// ---- VISUs/Behelyezes.TcVIS
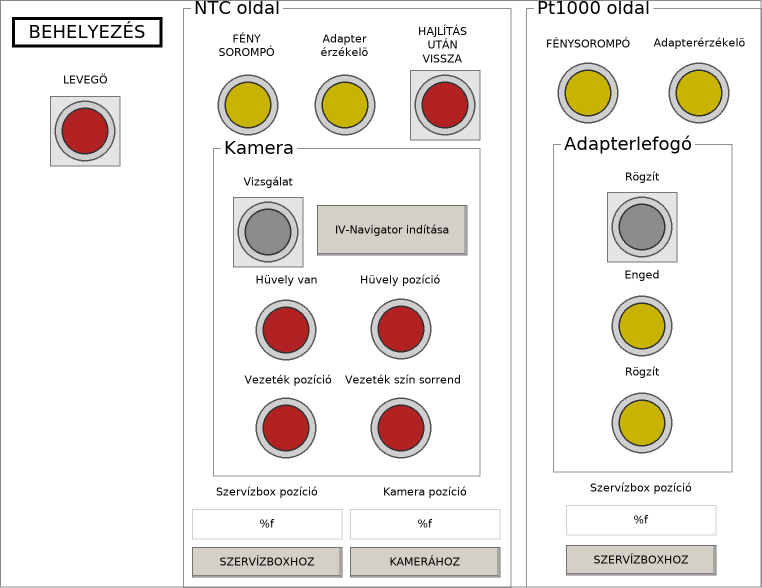
VISUALIZATION Behelyezes  // 762x588
    GroupBox (526,0 236x587), "Pt1000 oldal"
        GroupBox (27,136 179x336), "Adapterlefogó"
            PushSwitch (54,56 70x70), variable: GVL.bAdapterLefogo, behaviour: TOGGLE, style: Switch-PushSwitch-Gray
            Lamp1 (54,155 70x70), variable: GVL.bAdapterLefogoBent, style: Lamp-Lamp1-Yellow
            Lamp1 (54,252 70x70), variable: GVL.bAdapterLefogoKint, style: Lamp-Lamp1-Yellow
            Label (61,226 57x20), "Rögzít"
            Label (62,129 54x20), "Enged"
            Label (60,31 59x20), "Rögzít"
        Lamp1 (138,58 70x70), variable: GVL.bAdaptererzekelo, style: Lamp-Lamp1-Yellow
        Label (122,33 103x20), "Adapterérzékelö"
        Lamp1 (27,58 70x70), variable: GVL.bFenysorompoPt, style: Lamp-Lamp1-Yellow
        Label (10,34 104x20), "FÉNYSOROMPÓ"
        Group (40,478 150x97)
            Button (0,67 150x30), "SZERVÍZBOXHOZ"
                OnMouseUp: execute { PISTITENGELY.lrPistiPosition:=GVL.lrPtSzervizbox; PISTITENGELY.sPistiAxisCommand:='MOVE'; }
            Textfield (0,27 150x30), "%f", text variable: GVL.lrPtSzervizbox
                OnMouseClick: write the text variable via VisuDialogs.Numpad, min -10000, max -1
            Label (0,0 150x20), "Szervízbox pozíció"
    RoundedRectangle (12,17 150x30)
    Label (12,17 150x30), "BEHELYEZÉS"
    GroupBox (183,0 328x588), "NTC oldal"
        GroupBox (30,140 267x336), "Kamera"
            Group (20,32 70x95)
                PushSwitch (0,25 70x70), variable: GVL.bKameraTrigger, behaviour: TOGGLE, style: Switch-PushSwitch-Gray
                Label (2,0 67x20), "Vizsgálat"
            Lamp1 (153,154 70x70), variable: GVL.bKameraHulsePozOK, style: Lamp-Lamp1-Green
            Lamp1 (153,253 70x70), variable: GVL.bKameraSzinekOK, style: Lamp-Lamp1-Green
            Label (130,230 120x20), "Vezeték szín sorrend"
            Label (140,130 94x20), "Hüvely pozíció"
            Lamp1 (153,154 70x70), variable: NOT GVL.bKameraHulsePozOK, invisible if: NOT KAMERA.bVizsgalatKesz OR GVL.bKameraHulsePozOK, style: Lamp-Lamp1-Red
            Lamp1 (153,253 70x70), variable: NOT GVL.bKameraSzinekOK, invisible if: NOT KAMERA.bVizsgalatKesz OR GVL.bKameraSzinekOK, style: Lamp-Lamp1-Red
            Label (30,230 90x20), "Vezeték pozíció"
            Lamp1 (38,253 70x70), variable: GVL.bKameraVezetekPozOK, style: Lamp-Lamp1-Green
            Lamp1 (38,253 70x70), variable: NOT GVL.bKameraVezetekPozOK, invisible if: NOT KAMERA.bVizsgalatKesz OR GVL.bKameraVezetekPozOK, style: Lamp-Lamp1-Red
            Button (104,65 150x50), "IV-Navigator indítása", tooltip "A jelölö lézer saját vezérlö szoftvere", pressed state: Laser.bStartFOBADraw
                OnMouseUp: execute { KAMERA.bStartIVNav:=TRUE; }
            Label (32,130 83x20), "Hüvely van"
            Lamp1 (38,155 70x70), variable: GVL.bKameraHulseVanOK, style: Lamp-Lamp1-Green
            Lamp1 (38,155 70x70), variable: NOT GVL.bKameraHulseVanOK, invisible if: NOT KAMERA.bVizsgalatKesz OR GVL.bKameraHulseVanOK, style: Lamp-Lamp1-Red
        Group (9,482 150x95)
            Textfield (0,27 150x30), "%f", text variable: GVL.lrNTCSzervizbox
                OnMouseClick: write the text variable via VisuDialogs.Numpad, min -10000, max -1
            Button (0,65 150x30), "SZERVÍZBOXHOZ"
                OnMouseUp: execute { JOZSITENGELY.lrJozsiPosition:=GVL.lrNTCSzervizbox; JOZSITENGELY.sJozsiAxisCommand:='MOVE'; }
            Label (0,0 150x20), "Szervízbox pozíció"
        Lamp1 (30,70 70x70), variable: GVL.bFenysorompoNTC, style: Lamp-Lamp1-Yellow
        Label (10,30 107x31), "FÉNY SOROMPÓ"
        Group (167,482 150x95)
            Textfield (0,27 150x30), "%f", text variable: GVL.lrNTCKameraPosition
                OnMouseClick: write the text variable via VisuDialogs.Numpad, min -10000, max -1
            Button (0,65 150x30), "KAMERÁHOZ"
                OnMouseUp: execute { JOZSITENGELY.lrJozsiPosition:=GVL.lrNTCKameraPosition; JOZSITENGELY.sJozsiAxisCommand:='MOVE'; }
            Label (0,0 150x20), "Kamera pozíció"
        Label (110,30 103x31), "Adapter érzékelö"
        Label (220,20 79x50), "HAJLÍTÁS UTÁN VISSZA"
    Label (51,70 69x20), "LEVEGÖ"
    PushSwitch (50,96 70x70), variable: MAIN.bLevego, behaviour: TOGGLE, style: Switch-PushSwitch-Red
    Lamp1 (310,70 70x70), variable: GVL.bNTCAdapterErzekelo, style: Lamp-Lamp1-Yellow
    PushSwitch (410,70 70x70), variable: AUTOMATA.bHajlitasUtanVissza, behaviour: TOGGLE, style: Switch-PushSwitch-Red
END_VISUALIZATION

// ---- VISUs/Rendszerinditas.TcVIS
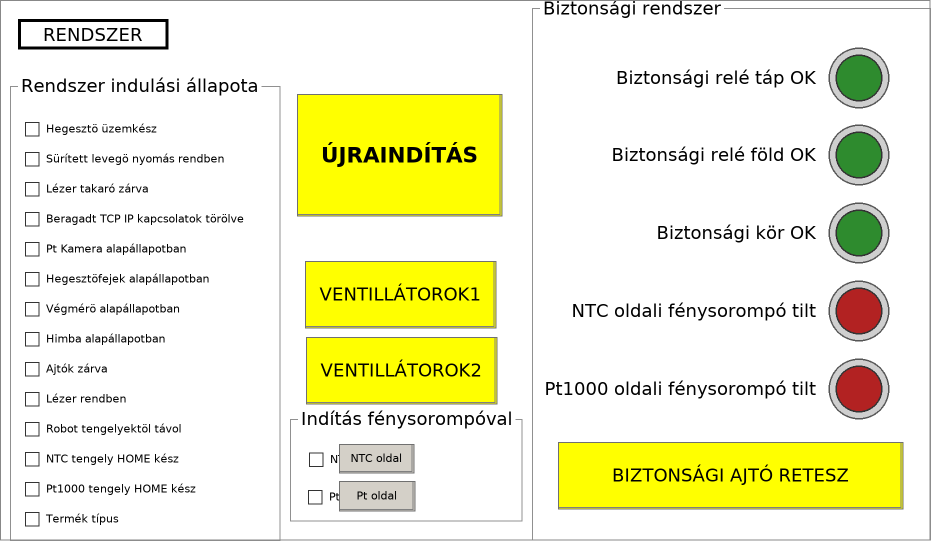
VISUALIZATION Rendszerinditas  // 931x541
    RoundedRectangle (18,19 150x30)
    Label (18,20 150x30), "RENDSZER"
    Button (297,94 205x122), "ÚJRAINDÍTÁS"
        OnMouseUp: execute { INIT.bRestart:=TRUE; }
    GroupBox (10,78 270x463), "Rendszer indulási állapota"
        Frame (13,36 239x351)
            shows Start_ellenorzes()
    GroupBox (532,0 399x540), "Biztonsági rendszer"
        Button (26,442 345x67), "BIZTONSÁGI AJTÓ RETESZ", pressed state: GVL.bBiztonsagiZarBe
            OnMouseClick: execute {
                IF GVL.bBiztonsagiZarBe=TRUE THEN
                	WHILE NOT (ROBOTREMOTE.sRobotCommand='') DO
                		;
                	END_WHILE
                	ROBOTREMOTE.sRobotCommand := 'Pause';
                	ROBOTREMOTE.bRobotCommandSend := TRUE;
                ELSE
                	WHILE NOT (ROBOTREMOTE.sRobotCommand='') DO
                		;
                	END_WHILE
                	ROBOTREMOTE.sRobotCommand := 'Continue';
                	ROBOTREMOTE.bRobotCommandSend := TRUE;
                END_IF
                GVL.bBiztonsagiZarBe:=NOT GVL.bBiztonsagiZarBe;
            }
        Lamp1 (292,43 70x70), variable: GVL.bBiztonsagiTap, style: Lamp-Lamp1-Green
        Label (17,63 270x30), "Biztonsági relé táp OK"
        Lamp1 (292,120 70x70), variable: NOT GVL.bBiztonsagiFold, style: Lamp-Lamp1-Green
        Label (17,140 270x30), "Biztonsági relé föld OK"
        Lamp1 (292,198 70x70), variable: (GVL.bBiztonsagiTap AND NOT GVL.bBiztonsagiFold) OR (NOT GVL.bBiztonsagiTap AND GVL.bBiztonsagiFold), style: Lamp-Lamp1-Green
        Label (17,218 270x30), "Biztonsági kör OK"
        Lamp1 (292,276 70x70), variable: NOT GVL.bFenysorompoNTC, style: Lamp-Lamp1-Red
        Label (17,296 270x30), "NTC oldali fénysorompó tilt"
        Lamp1 (292,354 70x70), variable: NOT GVL.bFenysorompoPt, style: Lamp-Lamp1-Red
        Label (17,374 270x30), "Pt1000 oldali fénysorompó tilt"
    Button (305,261 191x67), "VENTILLÁTOROK1", pressed state: GVL.bVentillatorok1Be
        toggle GVL.bVentillatorok1Be
    Button (306,337 191x67), "VENTILLÁTOROK2", pressed state: GVL.bVentillatorok2Be
        toggle GVL.bVentillatorok2Be
    GroupBox (290,411 232x110), "Indítás fénysorompóval"
        Checkbox (16,71 95x30), "Pt oldal", variable: GVL.bPtInditasFenysorompoval, input disabled if: TRUE
        Checkbox (17,34 94x29), "NTC oldal", variable: GVL.bNTCInditasFenysorompoval, input disabled if: TRUE
        Button (49,33 75x29), "NTC oldal", pressed state: GVL.bNTCInditasFenysorompoval
            toggle GVL.bNTCInditasFenysorompoval
            OnMouseUp: execute { AUTOMATA.iState:=102; }
        Button (49,70 76x30), "Pt oldal", pressed state: GVL.bPtInditasFenysorompoval
            toggle GVL.bPtInditasFenysorompoval
            OnMouseUp: execute { AUTOMATA.iState2:=103; }
END_VISUALIZATION

// ---- VISUs/Start_ellenorzes.TcVIS
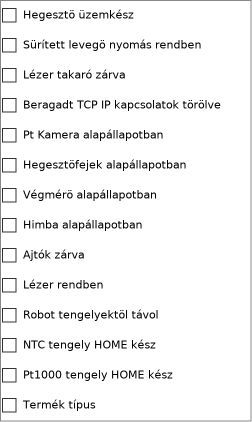
VISUALIZATION Start_ellenorzes  // 252x422
    Checkbox (0,30 250x30), "Sürített levegö nyomás rendben", variable: MAIN.bLevegoOK
    Checkbox (0,90 250x30), "Beragadt TCP IP kapcsolatok törölve", variable: INIT.bTCPKesz
    Checkbox (0,150 250x30), "Hegesztöfejek alapállapotban", variable: INIT.bHegesztoFejekKesz
    Checkbox (0,180 250x30), "Végmérö alapállapotban", variable: INIT.bVegmeroKesz
    Checkbox (0,300 250x30), "Robot tengelyektöl távol", variable: INIT.bRobotKesz
    Checkbox (0,270 250x30), "Lézer rendben", variable: INIT.bLezerKesz
    Checkbox (0,330 250x30), "NTC tengely HOME kész", variable: INIT.bNTCTengelyKesz
    Checkbox (0,360 250x30), "Pt1000 tengely HOME kész", variable: INIT.bPt1000TengelyKesz
    Checkbox (0,60 250x30), "Lézer takaró zárva", variable: VEGMERO.bLezertakaroZarva
    Checkbox (0,0 250x30), "Hegesztö üzemkész", variable: INIT.bHegesztoKesz
    Checkbox (0,390 250x30), "Termék típus", variable: GVL.bProductTypeOK
    Checkbox (0,240 250x30), "Ajtók zárva", variable: NOT GVL.bBiztonsagiFold AND GVL.bBiztonsagiTap
    Checkbox (0,210 250x30), "Himba alapállapotban", variable: INIT.bHimbaKesz
    Checkbox (0,120 250x30), "Pt Kamera alapállapotban", variable: INIT.bKameraKesz
END_VISUALIZATION

// ---- VISUs/Tengely_NTC_beallitasok.TcVIS
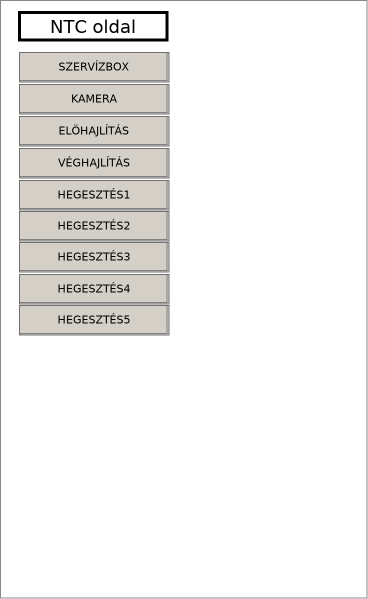
VISUALIZATION Tengely_NTC_beallitasok  // 368x599
    Label (297,567 69x30)
    RoundedRectangle (18,11 150x30)
    Label (18,12 150x30), "NTC oldal"
    Button (19,116 150x30), "ELÖHAJLÍTÁS"
        OnMouseUp: execute { GVL.iFoLapozo:=GVL.SZERVIZ_FUL; GVL.iSzervizLapozo:=GVL.HAJLITOK_FUL; }
    Button (19,148 150x30), "VÉGHAJLÍTÁS"
        OnMouseUp: execute { GVL.iFoLapozo:=GVL.SZERVIZ_FUL; GVL.iSzervizLapozo:=GVL.HAJLITOK_FUL; }
    Button (19,180 150x30), "HEGESZTÉS1"
        OnMouseUp: execute {
            GVL.iFoLapozo:=GVL.SZERVIZ_FUL;
            GVL.iSzervizLapozo:=GVL.HEGESZTES_FUL;
            GVL.iTengelyLapozo:=GVL.NTC_TENGELY_FUL;
        }
    Button (19,211 150x30), "HEGESZTÉS2"
        OnMouseUp: execute {
            GVL.iFoLapozo:=GVL.SZERVIZ_FUL;
            GVL.iSzervizLapozo:=GVL.HEGESZTES_FUL;
            GVL.iTengelyLapozo:=GVL.NTC_TENGELY_FUL;
        }
    Button (19,242 150x30), "HEGESZTÉS3"
        OnMouseUp: execute {
            GVL.iFoLapozo:=GVL.SZERVIZ_FUL;
            GVL.iSzervizLapozo:=GVL.HEGESZTES_FUL;
            GVL.iTengelyLapozo:=GVL.NTC_TENGELY_FUL;
        }
    Button (19,274 150x30), "HEGESZTÉS4"
        OnMouseUp: execute {
            GVL.iFoLapozo:=GVL.SZERVIZ_FUL;
            GVL.iSzervizLapozo:=GVL.HEGESZTES_FUL;
            GVL.iTengelyLapozo:=GVL.NTC_TENGELY_FUL;
        }
    Button (19,305 150x30), "HEGESZTÉS5"
        OnMouseUp: execute {
            GVL.iFoLapozo:=GVL.SZERVIZ_FUL;
            GVL.iSzervizLapozo:=GVL.HEGESZTES_FUL;
            GVL.iTengelyLapozo:=GVL.NTC_TENGELY_FUL;
        }
    Button (19,52 150x30), "SZERVÍZBOX"
        OnMouseUp: execute { GVL.iFoLapozo:=GVL.SZERVIZ_FUL; GVL.iSzervizLapozo:=GVL.BEHELYEZES_FUL; }
    Button (19,84 150x30), "KAMERA"
        OnMouseUp: execute { GVL.iFoLapozo:=GVL.SZERVIZ_FUL; GVL.iSzervizLapozo:=GVL.BEHELYEZES_FUL; }
END_VISUALIZATION

// ---- VISUs/Tengely_Pt1000.TcVIS
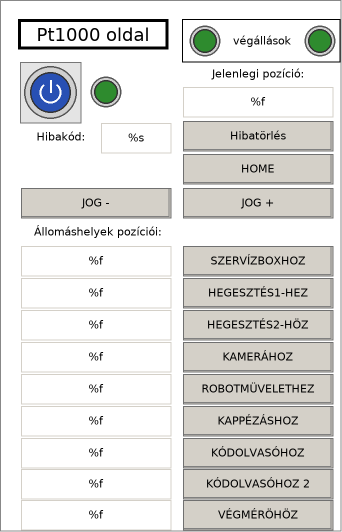
VISUALIZATION Tengely_Pt1000  // 342x532
    PowerSwitch (20,62 61x61), variable: GVL.bPistiServo, behaviour: TOGGLE, style: Switch-PowerSwitch-Blue
    Button (183,154 150x30), "HOME"
        OnMouseUp: execute { PISTITENGELY.sPistiAxisCommand:='HOME'; }
    Button (183,188 150x30), "JOG +"
        tap PISTITENGELY.bPistiJOGPlus
    Button (21,188 150x30), "JOG -"
        tap PISTITENGELY.bPistiJOGMinus
    Button (183,121 150x30), "Hibatörlés"
        tap PISTITENGELY.bPistiReset
    Textfield (101,123 70x30), "%s", text variable: PISTITENGELY.nPistiErrorCode, input disabled if: TRUE
    Textfield (21,310 150x30), "%f", text variable: GVL.lrHegesztoPosition7
    Button (183,310 150x30), "HEGESZTÉS2-HÖZ"
        OnMouseUp: execute { PISTITENGELY.lrPistiPosition:=GVL.lrHegesztoPosition7; PISTITENGELY.sPistiAxisCommand:='MOVE'; }
    Label (183,64 150x20), "Jelenlegi pozíció:"
    Textfield (183,87 150x30), "%f", text variable: PISTITENGELY.lrPistiActPos, input disabled if: TRUE
    Button (183,246 150x30), "SZERVÍZBOXHOZ"
        OnMouseUp: execute { PISTITENGELY.lrPistiPosition:=GVL.lrPtSzervizbox; PISTITENGELY.sPistiAxisCommand:='MOVE'; }
    Textfield (21,246 150x30), "%f", text variable: GVL.lrPtSzervizbox
    Textfield (21,278 150x30), "%f", text variable: GVL.lrHegesztoPosition6
    Button (183,278 150x30), "HEGESZTÉS1-HEZ"
        OnMouseUp: execute { PISTITENGELY.lrPistiPosition:=GVL.lrHegesztoPosition6; PISTITENGELY.sPistiAxisCommand:='MOVE'; }
    Lamp1 (88,74 36x36), variable: PISTITENGELY.bHomeReady, style: Lamp-Lamp1-Green
    RoundedRectangle (18,19 150x30)
    Label (18,20 150x30), "Pt1000 oldal"
    Textfield (21,374 150x30), "%f", text variable: GVL.lrRobotKappePosition
    Button (183,374 150x30), "ROBOTMÜVELETHEZ"
        OnMouseUp: execute { PISTITENGELY.lrPistiPosition:=GVL.lrRobotKappePosition; PISTITENGELY.sPistiAxisCommand:='MOVE'; }
    Textfield (21,500 150x30), "%f", text variable: GVL.lrVegmeroPosition
    Button (183,500 150x30), "VÉGMÉRÖHÖZ"
        OnMouseUp: execute { PISTITENGELY.lrPistiPosition:=GVL.lrVegmeroPosition; PISTITENGELY.sPistiAxisCommand:='MOVE'; }
    Textfield (21,406 150x30), "%f", text variable: GVL.lrKappePosition
    Button (183,406 150x30), "KAPPÉZÁSHOZ"
        OnMouseUp: execute { PISTITENGELY.lrPistiPosition:=GVL.lrKappePosition; PISTITENGELY.sPistiAxisCommand:='MOVE'; }
    Textfield (21,438 150x30), "%f", text variable: GVL.lrKodolvasasPosition
    Button (183,438 150x30), "KÓDOLVASÓHOZ"
        OnMouseUp: execute { PISTITENGELY.lrPistiPosition:=GVL.lrKodolvasasPosition; PISTITENGELY.sPistiAxisCommand:='MOVE'; }
    Label (26,127 70x20), "Hibakód:"
    Label (23,222 150x20), "Állomáshelyek pozíciói:"
    Group (182,19 158x43)
        Rectangle (0,0 158x43)
        Lamp1 (5,4 36x36), variable: GVL.bPistiNegSwitch, style: Lamp-Lamp1-Green
        Lamp1 (120,4 36x36), variable: GVL.bPistiPosSwitch, style: Lamp-Lamp1-Green
        Label (45,12 70x20), "végállások"
    Textfield (21,342 150x30), "%f", text variable: GVL.lrPtKameraPosition
    Button (183,342 150x30), "KAMERÁHOZ"
        OnMouseUp: execute { PISTITENGELY.lrPistiPosition:=GVL.lrPtKameraPosition; PISTITENGELY.sPistiAxisCommand:='MOVE'; }
    Textfield (21,469 150x30), "%f", text variable: GVL.lrKodolvasasPosition2
    Button (183,469 150x30), "KÓDOLVASÓHOZ 2"
        OnMouseUp: execute { PISTITENGELY.lrPistiPosition:=GVL.lrKodolvasasPosition2; PISTITENGELY.sPistiAxisCommand:='MOVE'; }
END_VISUALIZATION

// ---- VISUs/Tengelyek.TcVIS
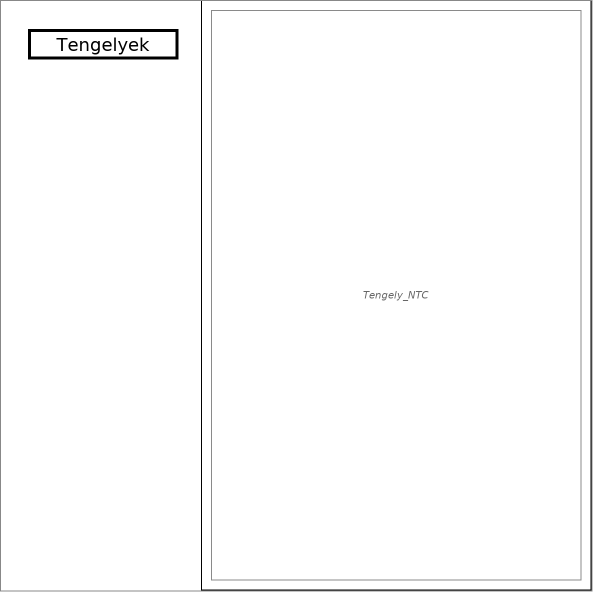
VISUALIZATION Tengelyek  // 593x592
    Group (201,0 390x590)
        Rectangle (0,0 390x590)
        TabControl (10,10 370x570)
            shows Tengely_NTC()
            shows Tengely_Pt1000()
            [0]: TabTitle=NTC oldal
            [1]: TabTitle=Pt1000 oldal
    RoundedRectangle (28,29 150x30)
    Label (28,30 150x30), "Tengelyek"
END_VISUALIZATION

// ---- VISUs/Tengely_NTC.TcVIS
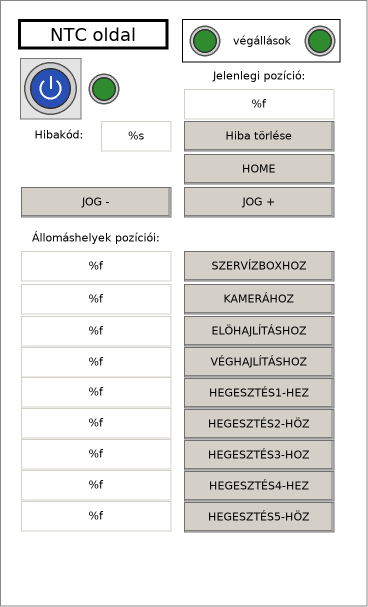
VISUALIZATION Tengely_NTC  // 368x607
    PowerSwitch (20,58 61x61), variable: GVL.bJozsiServo, behaviour: TOGGLE, style: Switch-PowerSwitch-Blue
    Button (184,154 150x30), "HOME"
        OnMouseUp: execute { JOZSITENGELY.sJozsiAxisCommand:='HOME'; }
    Button (184,187 150x30), "JOG +"
        tap JOZSITENGELY.bJozsiJOGPlus
    Button (21,187 150x30), "JOG -"
        tap JOZSITENGELY.bJozsiJOGMinus
    Button (184,121 150x30), "Hiba törlése"
        tap JOZSITENGELY.bJozsiReset
    Textfield (101,121 70x30), "%s", text variable: JOZSITENGELY.nJozsiErrorCode, input disabled if: TRUE
    Textfield (21,316 150x30), "%f", text variable: GVL.lrHajlitoPosition1
    Button (184,316 150x30), "ELÖHAJLÍTÁSHOZ"
        OnMouseUp: execute { JOZSITENGELY.lrJozsiPosition:=GVL.lrHajlitoPosition1; JOZSITENGELY.sJozsiAxisCommand:='MOVE'; }
    Textfield (184,89 150x30), "%f", text variable: JOZSITENGELY.lrJozsiActPos, input disabled if: TRUE
    Label (184,66 150x20), "Jelenlegi pozíció:"
    Textfield (21,284 150x30), "%f", text variable: GVL.lrNTCKameraPosition
    Button (184,284 150x30), "KAMERÁHOZ"
        OnMouseUp: execute { JOZSITENGELY.lrJozsiPosition:=GVL.lrNTCKameraPosition; JOZSITENGELY.sJozsiAxisCommand:='MOVE'; }
    Textfield (21,377 150x30), "%f", text variable: GVL.lrHegesztoPosition1
    Button (184,378 150x30), "HEGESZTÉS1-HEZ"
        OnMouseUp: execute { JOZSITENGELY.lrJozsiPosition:=GVL.lrHegesztoPosition1; JOZSITENGELY.sJozsiAxisCommand:='MOVE'; }
    Textfield (21,408 150x30), "%f", text variable: GVL.lrHegesztoPosition2
    Button (184,409 150x30), "HEGESZTÉS2-HÖZ"
        OnMouseUp: execute { JOZSITENGELY.lrJozsiPosition:=GVL.lrHegesztoPosition2; JOZSITENGELY.sJozsiAxisCommand:='MOVE'; }
    Textfield (21,439 150x30), "%f", text variable: GVL.lrHegesztoPosition3
    Button (184,440 150x30), "HEGESZTÉS3-HOZ"
        OnMouseUp: execute { JOZSITENGELY.lrJozsiPosition:=GVL.lrHegesztoPosition3; JOZSITENGELY.sJozsiAxisCommand:='MOVE'; }
    Textfield (21,470 150x30), "%f", text variable: GVL.lrHegesztoPosition4
    Button (184,471 150x30), "HEGESZTÉS4-HEZ"
        OnMouseUp: execute { JOZSITENGELY.lrJozsiPosition:=GVL.lrHegesztoPosition4; JOZSITENGELY.sJozsiAxisCommand:='MOVE'; }
    Textfield (21,501 150x30), "%f", text variable: GVL.lrHegesztoPosition5
    Button (184,502 150x30), "HEGESZTÉS5-HÖZ"
        OnMouseUp: execute { JOZSITENGELY.lrJozsiPosition:=GVL.lrHegesztoPosition5; JOZSITENGELY.sJozsiAxisCommand:='MOVE'; }
    Label (297,575 69x30)
    Button (184,251 150x30), "SZERVÍZBOXHOZ"
        OnMouseUp: execute { JOZSITENGELY.lrJozsiPosition:=GVL.lrNTCSzervizbox; JOZSITENGELY.sJozsiAxisCommand:='MOVE'; }
    Lamp1 (86,71 36x36), variable: JOZSITENGELY.bHomeReady, style: Lamp-Lamp1-Green
    Label (24,125 70x20), "Hibakód:"
    Label (21,228 150x20), "Állomáshelyek pozíciói:"
    RoundedRectangle (18,19 150x30)
    Label (18,20 150x30), "NTC oldal"
    Group (182,19 158x43)
        Rectangle (0,0 158x43)
        Lamp1 (5,4 36x36), variable: GVL.bJozsiNegSwitch, style: Lamp-Lamp1-Green
        Lamp1 (120,4 36x36), variable: GVL.bJozsiPosSwitch, style: Lamp-Lamp1-Green
        Label (45,12 70x20), "végállások"
    Textfield (21,251 150x30), "%f", text variable: GVL.lrNTCSzervizbox
    Textfield (21,347 150x30), "%f", text variable: GVL.lrHajlitoPosition2
    Button (184,347 150x30), "VÉGHAJLÍTÁSHOZ"
        OnMouseUp: execute { JOZSITENGELY.lrJozsiPosition:=GVL.lrHajlitoPosition2; JOZSITENGELY.sJozsiAxisCommand:='MOVE'; }
END_VISUALIZATION

// ---- VISUs/Tengely_Pt1000_beallitasok.TcVIS
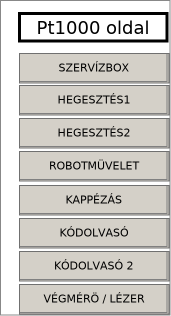
VISUALIZATION Tengely_Pt1000_beallitasok  // 171x316
    RoundedRectangle (18,12 150x30)
    Label (18,13 150x30), "Pt1000 oldal"
    Button (19,118 150x30), "HEGESZTÉS2"
        OnMouseUp: execute { GVL.iFoLapozo:=GVL.SZERVIZ_FUL; GVL.iSzervizLapozo:=GVL.HEGESZTES_FUL; }
    Button (19,53 150x30), "SZERVÍZBOX"
        OnMouseUp: execute {
            GVL.iFoLapozo:=GVL.SZERVIZ_FUL;
            GVL.iSzervizLapozo:=GVL.BEHELYEZES_FUL;
            GVL.iTengelyLapozo:=GVL.PT_TENGELY_FUL;
        }
    Button (19,85 150x30), "HEGESZTÉS1"
        OnMouseUp: execute { GVL.iFoLapozo:=GVL.SZERVIZ_FUL; GVL.iSzervizLapozo:=GVL.HEGESZTES_FUL; }
    Button (19,151 150x30), "ROBOTMÜVELET"
        OnMouseUp: execute { GVL.iFoLapozo:=GVL.SZERVIZ_FUL; GVL.iSzervizLapozo:=GVL.ROBOT_FUL; }
    Button (19,284 150x30), "VÉGMÉRÖ / LÉZER"
        OnMouseUp: execute { GVL.iFoLapozo:=GVL.SZERVIZ_FUL; GVL.iSzervizLapozo:=GVL.VEGMERO_FUL; }
    Button (19,185 150x30), "KAPPÉZÁS"
        OnMouseUp: execute { GVL.iFoLapozo:=GVL.SZERVIZ_FUL; GVL.iSzervizLapozo:=GVL.KAPPE_PRES_FUL; }
    Button (19,218 150x30), "KÓDOLVASÓ"
        OnMouseUp: execute { GVL.iFoLapozo:=GVL.SZERVIZ_FUL; GVL.iSzervizLapozo:=GVL.KODOLVASO_FUL; }
    Button (19,251 150x30), "KÓDOLVASÓ 2"
        OnMouseUp: execute { GVL.iFoLapozo:=GVL.SZERVIZ_FUL; GVL.iSzervizLapozo:=GVL.KODOLVASO_FUL; }
END_VISUALIZATION

// ---- VISUs/Termektipus.TcVIS
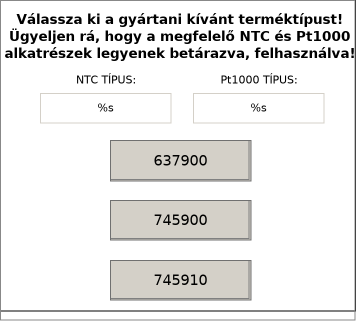
VISUALIZATION Termektipus  // 356x321
    RoundedRectangle (0,0 356x311)
    Label (51,70 110x20), "NTC TÍPUS:"
    Textfield (40,93 131x30), "%s", text variable: GVL.sNTCTypeElozo, colour toggle: GVL.sNTCType='HIBÁS KÓD', input disabled if: true
        OnMouseClick: write GVL.sNTCType via Edit
    Textfield (193,93 131x30), "%s", text variable: GVL.sPtTypeElozo, colour toggle: GVL.sPtType='HIBÁS KÓD', input disabled if: true
        OnMouseClick: write GVL.sPtType via Edit
    Label (204,70 110x20), "Pt1000 TÍPUS:"
    Textfield (120,150 131x30), "%s", text variable: GVL.sProductType, colour toggle: NOT GVL.bProductTypeOK, invisible if: true
        OnMouseClick: write the text variable via Edit
        OnMouseClick: CloseDialog Dialog=Termektipus, Result=OK, NumpadKeypadSet=True
    Button (110,140 141x41), "637900", input disabled if: GVL.UserActual.UserLevel<1
        OnMouseClick: execute { GVL.sProductType:='637900'; }
        OnMouseClick: CloseDialog Dialog=Termektipus, Result=OK, NumpadKeypadSet=True
    Button (110,200 141x40), "745900", input disabled if: GVL.UserActual.UserLevel<1
        OnMouseClick: execute { GVL.sProductType:='745900'; }
        OnMouseClick: CloseDialog Dialog=Termektipus, Result=OK, NumpadKeypadSet=True
    Button (110,260 141x40), "745910", input disabled if: GVL.UserActual.UserLevel<1
        OnMouseClick: execute { GVL.sProductType:='745910'; }
        OnMouseClick: CloseDialog Dialog=Termektipus, Result=OK, NumpadKeypadSet=True
    Label (10,-10 340x93), "Válassza ki a gyártani kívánt terméktípust! Ügyeljen rá, hogy a megfelelő NTC és Pt1000 alkatrészek legyenek betárazva, felhasználva!"
END_VISUALIZATION

// ---- VISUs/Vegmero.TcVIS
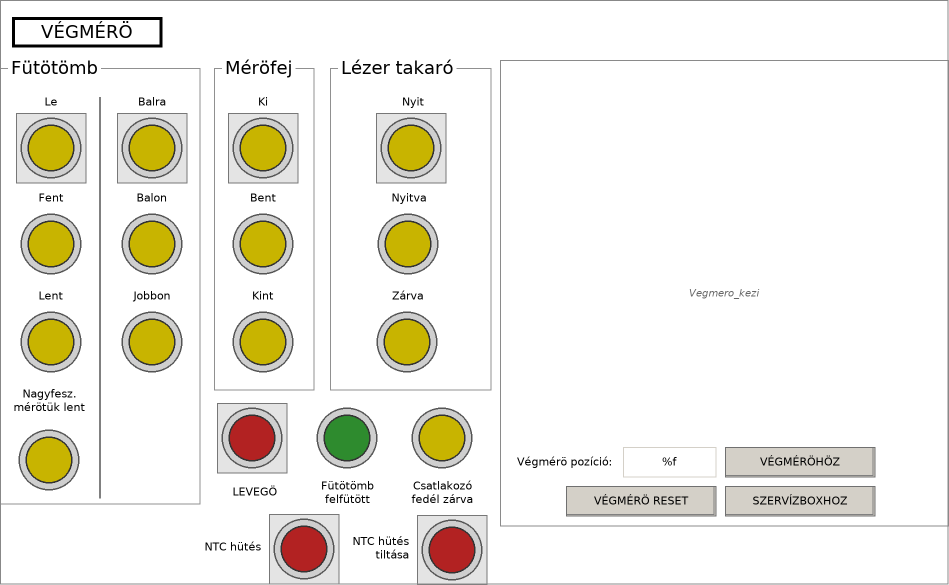
VISUALIZATION Vegmero  // 949x585
    Lamp1 (407,403 70x70), variable: VEGMERO.bFedelNyitva, style: Lamp-Lamp1-Yellow
    Label (405,478 75x29), "Csatlakozó fedél zárva"
    GroupBox (0,60 200x444), "Fütötömb"
        Lamp1 (16,247 70x70), variable: VEGMERO.bPlatniLent, style: Lamp-Lamp1-Yellow
        Label (26,226 50x20), "Lent"
        PushSwitch (16,53 70x70), variable: VEGMERO.bPlatniFelLe, behaviour: TOGGLE, style: Switch-PushSwitch-Yellow
        Label (26,32 50x20), "Le"
        Lamp1 (16,149 70x70), variable: VEGMERO.bPlatniFent, style: Lamp-Lamp1-Yellow
        Label (26,128 50x20), "Fent"
        Lamp1 (117,149 70x70), variable: VEGMERO.bPlatniBalon, style: Lamp-Lamp1-Yellow
        Label (127,128 50x20), "Balon"
        Lamp1 (117,247 70x70), variable: VEGMERO.bPlatniJobbon, style: Lamp-Lamp1-Yellow
        Label (127,226 50x20), "Jobbon"
        PushSwitch (117,53 70x70), variable: VEGMERO.bPlatniBalraJobbra, behaviour: TOGGLE, style: Switch-PushSwitch-Yellow
        Label (127,32 50x20), "Balra"
        Line (100,438) (100,37)
        Label (8,323 83x35), "Nagyfesz. mérötük lent"
        Lamp1 (14,365 70x70), variable: VEGMERO.bNagyFeszMerotuLent, style: Lamp-Lamp1-Yellow
    GroupBox (214,60 100x330), "Méröfej"
        Lamp1 (14,149 70x70), variable: VEGMERO.bMerotukBent, style: Lamp-Lamp1-Yellow
        Label (24,128 50x20), "Bent"
        Lamp1 (14,247 70x70), variable: VEGMERO.bMerotukKint, style: Lamp-Lamp1-Yellow
        Label (24,226 50x20), "Kint"
        PushSwitch (14,53 70x70), variable: VEGMERO.bMerotukBeKi, behaviour: TOGGLE, style: Switch-PushSwitch-Yellow
        Label (24,32 50x20), "Ki"
    GroupBox (330,60 161x330), "Lézer takaró"
        PushSwitch (46,53 70x70), variable: VEGMERO.bLezertakaro, behaviour: TOGGLE, style: Switch-PushSwitch-Yellow
        Label (58,32 50x20), "Nyit"
        Lamp1 (43,149 70x70), variable: VEGMERO.bLezertakaroNyitva, style: Lamp-Lamp1-Yellow
        Label (54,128 50x20), "Nyitva"
        Lamp1 (42,247 70x70), variable: VEGMERO.bLezertakaroZarva, style: Lamp-Lamp1-Yellow
        Label (53,226 50x20), "Zárva"
    TabControl (500,60 449x466)
        shows Vegmero_kezi()
        shows Vegmero_auto()
        [0]: TabTitle=Kézi
        [1]: TabTitle=Automata
    RoundedRectangle (12,17 150x30)
    Label (12,17 150x30), "VÉGMÉRÖ"
    Label (511,452 104x20), "Végmérö pozíció:"
    Textfield (623,447 93x30), "%f", text variable: GVL.lrVegmeroPosition
        OnMouseClick: write the text variable via VisuDialogs.Numpad, min -10000, max -1
    Button (725,447 150x30), "VÉGMÉRÖHÖZ"
        OnMouseUp: execute { PISTITENGELY.lrPistiPosition:=GVL.lrVegmeroPosition; PISTITENGELY.sPistiAxisCommand:='MOVE'; }
    Lamp1 (312,403 70x70), variable: GVL.bHeatingTempOK, style: Lamp-Lamp1-Green
    Label (310,478 75x29), "Fütötömb felfütött"
    Group (217,403 70x104)
        PushSwitch (0,0 70x70), variable: MAIN.bLevego, behaviour: TOGGLE, style: Switch-PushSwitch-Red
        Label (8,74 55x30), "LEVEGÖ"
    Button (725,486 150x30), "SZERVÍZBOXHOZ"
        OnMouseUp: execute { PISTITENGELY.lrPistiPosition:=GVL.lrPtSzervizbox; PISTITENGELY.sPistiAxisCommand:='MOVE'; }
    Button (566,486 150x30), "VÉGMÉRÖ RESET"
        OnMouseUp: execute { VEGMERO.iState:=0; VEGMERO.s_InCommand:='RESET'; }
    PushSwitch (269,514 70x70), variable: VEGMERO.bKeziHutes, behaviour: TOGGLE, style: Switch-PushSwitch-Red
    Label (196,532 68x30), "NTC hütés"
    PushSwitch (417,515 70x70), variable: VEGMERO.bHutesTiltas, behaviour: TOGGLE, style: Switch-PushSwitch-Red
    Label (344,533 68x30), "NTC hütés tiltása"
END_VISUALIZATION

// ---- VISUs/Hegesztes_Tengely_Pt1000.TcVIS
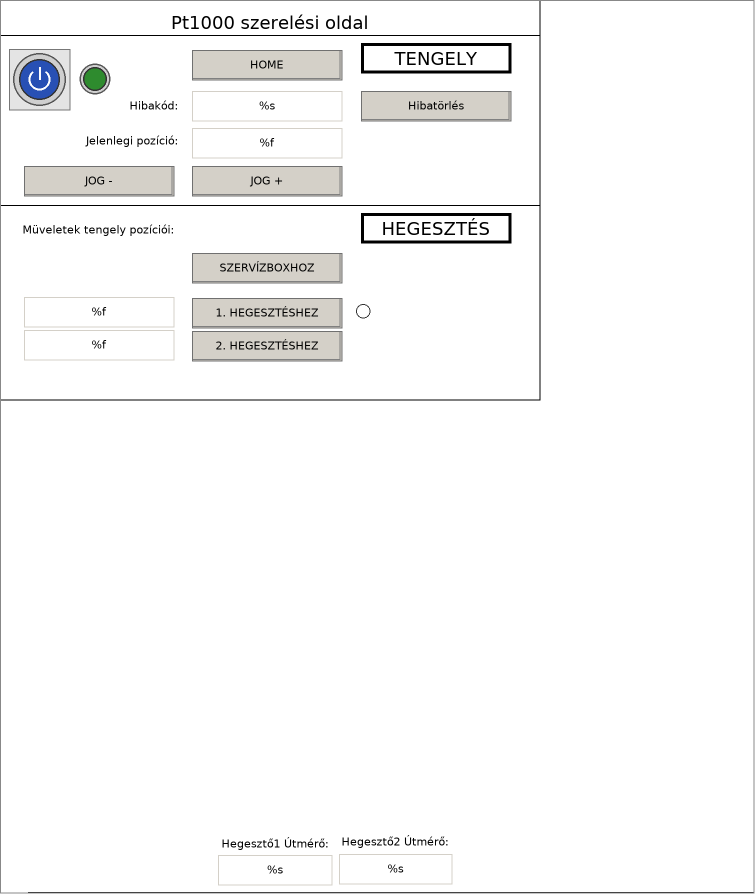
VISUALIZATION Hegesztes_Tengely_Pt1000  // 755x894
    Rectangle (0,0 540x400)
    Line (0,205) (540,205)
    Line (0,35) (540,35), "Pt1000 szerelési oldal"
    PowerSwitch (9,49 61x61), variable: GVL.bPistiServo, behaviour: TOGGLE, style: Switch-PowerSwitch-Blue
    Button (192,50 150x30), "HOME"
        OnMouseUp: execute { PISTITENGELY.sPistiAxisCommand:='HOME'; }
    Button (192,166 150x30), "JOG +"
        tap PISTITENGELY.bPistiJOGPlus
    Button (24,166 150x30), "JOG -"
        tap PISTITENGELY.bPistiJOGMinus
    Button (361,91 150x30), "Hibatörlés"
        tap PISTITENGELY.bPistiReset
    Textfield (192,91 150x30), "%s", text variable: PISTITENGELY.nPistiErrorCode, input disabled if: TRUE
    Textfield (24,330 150x30), "%f", text variable: GVL.lrHegesztoPosition7
        OnMouseClick: write the text variable via VisuDialogs.Numpad, min -10000, max -1
    Button (192,331 150x30), "2. HEGESZTÉSHEZ"
        OnMouseUp: execute { PISTITENGELY.lrPistiPosition:=GVL.lrHegesztoPosition7; PISTITENGELY.sPistiAxisCommand:='MOVE'; }
    Label (70,126 111x30), "Jelenlegi pozíció:"
    Textfield (192,128 150x30), "%f", text variable: PISTITENGELY.lrPistiActPos, input disabled if: TRUE
    RadioButton (354,253 170x116), variable: HEGESZTOK.nHegesztoNum
        Areas[0]: Text=Készenléti program
        Areas[6]: Text=6. hegesztés program
        Areas[7]: Text=7. hegesztés program
    Textfield (218,855 114x30), "%s", text variable: HEGESZTOK.ulHegeszto1Utmero, input disabled if: TRUE
    Label (200,829 150x30), "Hegesztő1 Útmérő:"
    Textfield (339,854 113x30), "%s", text variable: HEGESZTOK.ulHegeszto2Utmero, input disabled if: TRUE
    Label (320,827 150x30), "Hegesztő2 Útmérő:"
    Line (28,892) (753,892)
    Button (192,253 150x30), "SZERVÍZBOXHOZ"
        OnMouseUp: execute { PISTITENGELY.lrPistiPosition:=GVL.lrPtSzervizbox; PISTITENGELY.sPistiAxisCommand:='MOVE'; }
    Textfield (24,297 150x30), "%f", text variable: GVL.lrHegesztoPosition6
        OnMouseClick: write the text variable via VisuDialogs.Numpad, min -10000, max -1
    Button (192,298 150x30), "1. HEGESZTÉSHEZ"
        OnMouseUp: execute { PISTITENGELY.lrPistiPosition:=GVL.lrHegesztoPosition6; PISTITENGELY.sPistiAxisCommand:='MOVE'; }
    Lamp1 (77,61 36x36), variable: PISTITENGELY.bHomeReady, style: Lamp-Lamp1-Green
    Label (117,91 64x30), "Hibakód:"
    RoundedRectangle (361,43 150x30)
    Label (361,44 150x30), "TENGELY"
    RoundedRectangle (361,213 150x30)
    Label (361,214 150x30), "HEGESZTÉS"
    Label (17,215 163x30), "Müveletek tengely pozíciói:"
END_VISUALIZATION

// ---- VISUs/Hegesztes_Tengely_NTC.TcVIS
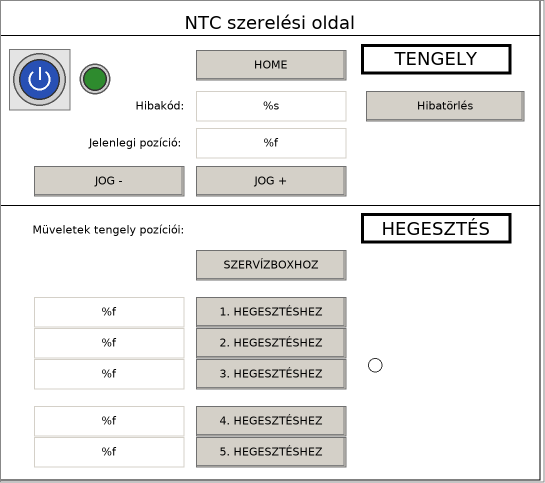
VISUALIZATION Hegesztes_Tengely_NTC  // 545x483
    Rectangle (0,0 540x480)
    PowerSwitch (9,49 61x61), variable: GVL.bJozsiServo, behaviour: TOGGLE, style: Switch-PowerSwitch-Blue
    Button (196,50 150x30), "HOME"
        OnMouseUp: execute { JOZSITENGELY.sJozsiAxisCommand:='HOME'; }
    Button (196,166 150x30), "JOG +"
        tap JOZSITENGELY.bJozsiJOGPlus
    Button (34,166 150x30), "JOG -"
        tap JOZSITENGELY.bJozsiJOGMinus
    Button (366,91 158x30), "Hibatörlés"
        tap JOZSITENGELY.bJozsiReset
    Textfield (196,91 150x30), "%s", text variable: JOZSITENGELY.nJozsiErrorCode, input disabled if: TRUE
    Label (34,128 150x30), "Jelenlegi pozíció:"
    Textfield (196,128 150x30), "%f", text variable: JOZSITENGELY.lrJozsiActPos, input disabled if: TRUE
    Textfield (34,297 150x30), "%f", text variable: GVL.lrHegesztoPosition1
        OnMouseClick: write the text variable via VisuDialogs.Numpad, min -10000, max -1
    Button (196,297 150x30), "1. HEGESZTÉSHEZ"
        OnMouseUp: execute { JOZSITENGELY.lrJozsiPosition:=GVL.lrHegesztoPosition1; JOZSITENGELY.sJozsiAxisCommand:='MOVE'; }
    RadioButton (366,249 177x232), variable: HEGESZTOK.nHegesztoNum
        Areas[0]: Text=Semelyik
        Areas[1]: Text=Program1HG1
        Areas[2]: Text=Program2HG1
        Areas[3]: Text=Program3HG1
        Areas[4]: Text=Program4HG2
        Areas[5]: Text=Program5HG2
        p340057476: Készenléti program
        p3123465237: 1. hegesztés program
        p2481256679: 2. hegesztés program
        p1032612214: 3. hegesztés program
        p3228930307: 4. hegesztés program
        p1847394450: 5. hegesztés program
        p1205187680: Program7HG3
        p3921487345: Program8HG3
    Textfield (34,328 150x30), "%f", text variable: GVL.lrHegesztoPosition2
        OnMouseClick: write the text variable via VisuDialogs.Numpad, min -10000, max -1
    Button (196,328 150x30), "2. HEGESZTÉSHEZ"
        OnMouseUp: execute { JOZSITENGELY.lrJozsiPosition:=GVL.lrHegesztoPosition2; JOZSITENGELY.sJozsiAxisCommand:='MOVE'; }
    Textfield (34,359 150x30), "%f", text variable: GVL.lrHegesztoPosition3
        OnMouseClick: write the text variable via VisuDialogs.Numpad, min -10000, max -1
    Button (196,359 150x30), "3. HEGESZTÉSHEZ"
        OnMouseUp: execute { JOZSITENGELY.lrJozsiPosition:=GVL.lrHegesztoPosition3; JOZSITENGELY.sJozsiAxisCommand:='MOVE'; }
    Textfield (34,406 150x30), "%f", text variable: GVL.lrHegesztoPosition4
        OnMouseClick: write the text variable via VisuDialogs.Numpad, min -10000, max -1
    Button (196,406 150x30), "4. HEGESZTÉSHEZ"
        OnMouseUp: execute { JOZSITENGELY.lrJozsiPosition:=GVL.lrHegesztoPosition4; JOZSITENGELY.sJozsiAxisCommand:='MOVE'; }
    Textfield (34,437 150x30), "%f", text variable: GVL.lrHegesztoPosition5
        OnMouseClick: write the text variable via VisuDialogs.Numpad, min -10000, max -1
    Button (196,437 150x30), "5. HEGESZTÉSHEZ"
        OnMouseUp: execute { JOZSITENGELY.lrJozsiPosition:=GVL.lrHegesztoPosition5; JOZSITENGELY.sJozsiAxisCommand:='MOVE'; }
    Button (196,250 150x30), "SZERVÍZBOXHOZ"
        OnMouseUp: execute { JOZSITENGELY.lrJozsiPosition:=GVL.lrNTCSzervizbox; JOZSITENGELY.sJozsiAxisCommand:='MOVE'; }
    Lamp1 (77,61 36x36), variable: JOZSITENGELY.bHomeReady, style: Lamp-Lamp1-Green
    Line (0,35) (540,35), "NTC szerelési oldal"
    Label (127,91 60x30), "Hibakód:"
    Line (0,205) (540,205)
    RoundedRectangle (361,44 150x30)
    Label (361,44 150x30), "TENGELY"
    RoundedRectangle (361,213 150x30)
    Label (361,214 150x30), "HEGESZTÉS"
    Label (27,215 163x30), "Müveletek tengely pozíciói:"
END_VISUALIZATION

// ---- VISUs/Kodolvaso.TcVIS
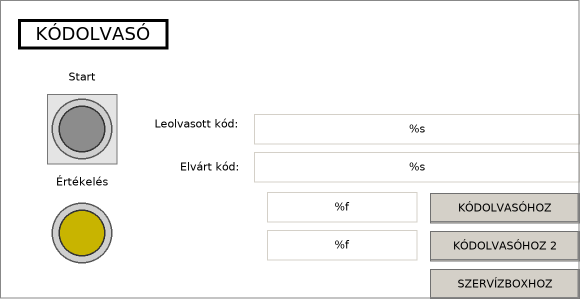
VISUALIZATION Kodolvaso  // 580x299
    PushSwitch (47,94 70x70), variable: ZEBRASCANNER.bStartSend, behaviour: TOGGLE, style: Switch-PushSwitch-Gray
    Lamp1 (47,198 70x70), variable: GVL.bMarkingOK, style: Lamp-Lamp1-Yellow
    Textfield (254,114 326x30), "%s", text variable: ZEBRASCANNER.sReceivedString255
    Label (48,67 68x20), "Start"
    Label (48,172 68x20), "Értékelés"
    Label (149,114 92x20), "Leolvasott kód:"
    Label (150,157 92x20), "Elvárt kód:"
    Textfield (254,152 326x30), "%s", text variable: ZEBRASCANNER.sExpectedString
    RoundedRectangle (18,19 150x30)
    Label (18,19 150x30), "KÓDOLVASÓ"
    Textfield (267,192 150x30), "%f", text variable: GVL.lrKodolvasasPosition
        OnMouseClick: write the text variable via VisuDialogs.Numpad, min -10000, max -1
    Button (430,193 150x30), "KÓDOLVASÓHOZ"
        OnMouseUp: execute { PISTITENGELY.lrPistiPosition:=GVL.lrKodolvasasPosition; PISTITENGELY.sPistiAxisCommand:='MOVE'; }
    Button (430,269 150x30), "SZERVÍZBOXHOZ"
        OnMouseUp: execute { PISTITENGELY.lrPistiPosition:=GVL.lrPtSzervizbox; PISTITENGELY.sPistiAxisCommand:='MOVE'; }
    Textfield (267,230 150x30), "%f", text variable: GVL.lrKodolvasasPosition2
        OnMouseClick: write the text variable via VisuDialogs.Numpad, min -10000, max -1
    Button (430,231 150x30), "KÓDOLVASÓHOZ 2"
        OnMouseUp: execute { PISTITENGELY.lrPistiPosition:=GVL.lrKodolvasasPosition2; PISTITENGELY.sPistiAxisCommand:='MOVE'; }
END_VISUALIZATION

// ---- VISUs/Hajlitok.TcVIS
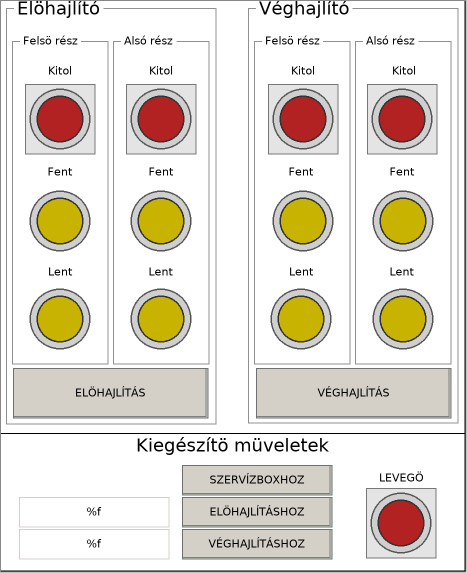
VISUALIZATION Hajlitok  // 467x573
    Rectangle (0,0 465x571)
    GroupBox (6,0 210x424), "Elöhajlító"
        GroupBox (6,33 96x331), "Felsö rész"
            PushSwitch (13,51 70x70), variable: HAJLITOK.bElohajlitoFelso, behaviour: TOGGLE, style: Switch-PushSwitch-Red
            Label (14,23 68x30), "Kitol"
            Lamp1 (13,153 70x70), variable: HAJLITOK.bElohajlitoFelsoFent, style: Lamp-Lamp1-Yellow
            Label (27,124 42x30), "Fent"
            Lamp1 (13,251 70x70), variable: HAJLITOK.bElohajlitoFelsoLent, style: Lamp-Lamp1-Yellow
            Label (29,224 39x30), "Lent"
        GroupBox (107,33 96x331), "Alsó rész"
            Label (14,23 68x30), "Kitol"
            Label (27,124 42x30), "Fent"
            PushSwitch (13,51 70x70), variable: HAJLITOK.bElohajlitoAlso, behaviour: TOGGLE, style: Switch-PushSwitch-Red
            Lamp1 (13,153 70x70), variable: HAJLITOK.bElohajlitoAlsoFent, style: Lamp-Lamp1-Yellow
            Lamp1 (13,251 70x70), variable: HAJLITOK.bElohajlitoAlsoLent, style: Lamp-Lamp1-Yellow
            Label (28,224 40x30), "Lent"
        Button (7,368 195x50), "ELÖHAJLÍTÁS", input disabled if: HAJLITOK.s_InCommand <> ''
            OnMouseUp: execute {
                IF HAJLITOK.s_InCommand = '' THEN
                	HAJLITOK.s_InCommand:='ELOHAJLITAS';
                END_IF
            }
    GroupBox (248,0 210x423), "Véghajlító"
        GroupBox (6,33 96x331), "Felsö rész"
            Label (15,23 68x30), "Kitol"
            Label (26,124 42x30), "Fent"
            Label (28,224 39x30), "Lent"
            PushSwitch (14,51 70x70), variable: HAJLITOK.bVeghajlitoFelso, behaviour: TOGGLE, style: Switch-PushSwitch-Red
            Lamp1 (14,153 70x70), variable: HAJLITOK.bVeghajlitoFelsoFent, style: Lamp-Lamp1-Yellow
            Lamp1 (12,251 70x70), variable: HAJLITOK.bVeghajlitoFelsoLent, style: Lamp-Lamp1-Yellow
        GroupBox (107,33 96x331), "Alsó rész"
            Label (15,23 68x30), "Kitol"
            Label (26,124 42x30), "Fent"
            Label (27,224 40x30), "Lent"
            PushSwitch (12,51 70x70), variable: HAJLITOK.bVeghajlitoAlso, behaviour: TOGGLE, style: Switch-PushSwitch-Red
            Lamp1 (13,153 70x70), variable: HAJLITOK.bVeghajlitoAlsoFent, style: Lamp-Lamp1-Yellow
            Lamp1 (13,251 70x70), variable: HAJLITOK.bVeghajlitoAlsoLent, style: Lamp-Lamp1-Yellow
        Button (8,368 195x50), "VÉGHAJLÍTÁS", input disabled if: HAJLITOK.s_InCommand <> ''
            OnMouseUp: execute {
                IF HAJLITOK.s_InCommand = '' THEN
                	HAJLITOK.s_InCommand:='VEGHAJLITAS';
                END_IF
            }
    Line (0,433) (465,433), "Kiegészítö müveletek"
    Textfield (19,497 150x30), "%f", text variable: GVL.lrHajlitoPosition1
        OnMouseClick: write the text variable via VisuDialogs.Numpad, min -10000, max -1
    Button (182,497 150x30), "ELÖHAJLÍTÁSHOZ", text variable: GVL.lrHajlitoPosition1
        OnMouseUp: execute { JOZSITENGELY.lrJozsiPosition:=GVL.lrHajlitoPosition1; JOZSITENGELY.sJozsiAxisCommand:='MOVE'; }
    Textfield (19,529 150x30), "%f", text variable: GVL.lrHajlitoPosition2
        OnMouseClick: write the text variable via VisuDialogs.Numpad, min -10000, max -1
    Button (182,529 150x30), "VÉGHAJLÍTÁSHOZ"
        OnMouseUp: execute { JOZSITENGELY.lrJozsiPosition:=GVL.lrHajlitoPosition2; JOZSITENGELY.sJozsiAxisCommand:='MOVE'; }
    Button (182,465 150x30), "SZERVÍZBOXHOZ"
        OnMouseUp: execute { JOZSITENGELY.lrJozsiPosition:=GVL.lrNTCSzervizbox; JOZSITENGELY.sJozsiAxisCommand:='MOVE'; }
    Group (366,463 70x95)
        PushSwitch (0,25 70x70), variable: MAIN.bLevego, behaviour: TOGGLE, style: Switch-PushSwitch-Red
        Label (1,0 69x30), "LEVEGÖ"
END_VISUALIZATION

// ---- VISUs/Szerviz.TcVIS
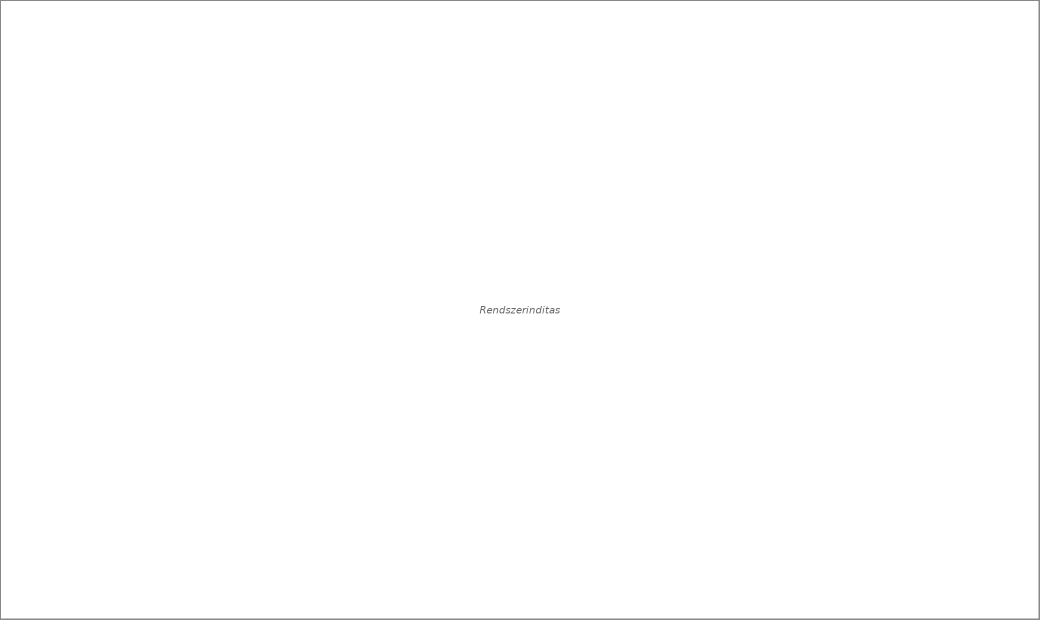
VISUALIZATION Szerviz  // 1040x620
    TabControl (0,0 1040x620), invisible if: GVL.UserActual.UserLevel<2, frame switch variable: GVL.iSzervizLapozo
        shows Rendszerinditas()
        shows Behelyezes()
        shows Tengelyek()
        shows Hajlitok()
        shows Hegesztok()
        shows Robot()
        shows NTC_szerviz()
        shows Kappe_pres()
        shows Vegmero()
        shows Lezer()
        shows Kodolvaso()
        shows Himba()
        shows Kamera_Pt()
        [0]: TabTitle=Rendszer
        [1]: TabTitle=Behelyezés
        [2]: TabTitle=Tengelyek
        [3]: TabTitle=Hajlítók
        [4]: TabTitle=Hegesztés
        [5]: TabTitle=Robot
        [6]: TabTitle=NTC vágó
        [7]: TabTitle=Kappe prés
        [8]: TabTitle=Végmérö
        [9]: TabTitle=Lézer
        [10]: TabTitle=Kódolvasó
        [11]: TabTitle=Himba
        [12]: TabTitle=Kamera Pt
END_VISUALIZATION

// ---- VISUs/NTC_szerviz.TcVIS
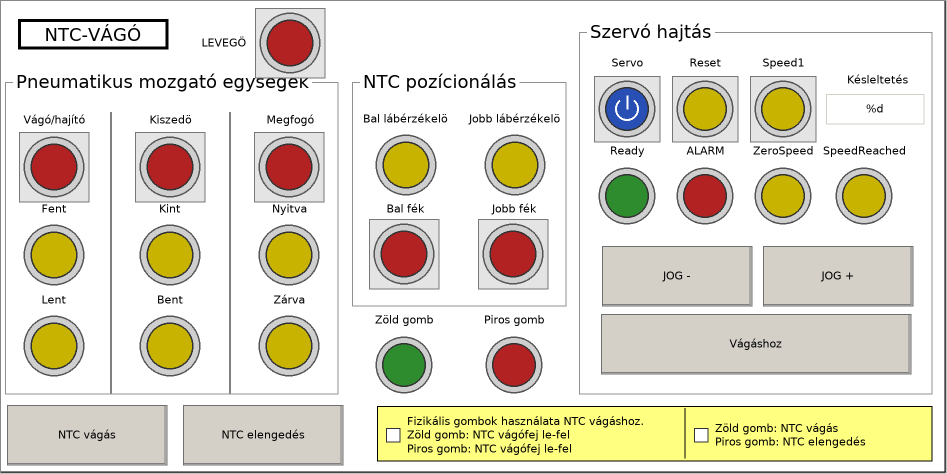
VISUALIZATION NTC_szerviz  // 947x474
    Rectangle (0,0 945x472)
    GroupBox (579,24 353x370), "Szervó hajtás"
        Lamp1 (15,139 66x66), variable: NTC.bReady, style: Lamp-Lamp1-Green
        Lamp1 (93,139 66x66), variable: NTC.bAlarm, style: Lamp-Lamp1-Red
        PowerSwitch (15,52 66x66), variable: NTC.bServoON, behaviour: TOGGLE, style: Switch-PowerSwitch-Blue
        PushSwitch (93,52 66x66), variable: NTC.bReset, behaviour: TOGGLE, style: Switch-PushSwitch-Yellow
        Lamp1 (171,139 66x66), variable: NTC.bZeroSpeed, style: Lamp-Lamp1-Yellow
        Label (170,112 69x30), "ZeroSpeed"
        Lamp1 (252,139 66x66), variable: NTC.bSpeedReached, style: Lamp-Lamp1-Yellow
        Label (239,112 93x30), "SpeedReached"
        PushSwitch (171,52 66x66), variable: NTC.bSpeed1, behaviour: TOGGLE, style: Switch-PushSwitch-Yellow
        Label (170,24 69x30), "Speed1"
        Button (184,222 150x60), "JOG +"
            tap NTC.bJogPlus
        Button (23,222 150x60), "JOG -"
            tap NTC.bJogMinus
        Textfield (247,70 98x30), "%d", text variable: NTC.iDelayFor
            OnMouseClick: write the text variable via VisuDialogs.Numpad, min -10000, max -1
        Label (264,41 69x30), "Késleltetés"
        Button (22,290 310x60), "Vágáshoz"
            OnMouseClick: execute { NTC.bVagashoz:=TRUE; }
        Label (14,24 69x30), "Servo"
        Label (92,24 69x30), "Reset"
        Label (14,112 69x30), "Ready"
        Label (92,112 69x30), "ALARM"
    GroupBox (5,74 333x320), "Pneumatikus mozgató egységek"
        PushSwitch (14,58 70x70), variable: NTCProcess.bVagoHajlito, behaviour: TOGGLE, style: Switch-PushSwitch-Red
        Label (15,31 69x30), "Vágó/hajító"
        Lamp1 (14,237 70x70), variable: NTCProcess.bVagoHajlitoLent, style: Lamp-Lamp1-Yellow
        Label (27,211 44x30), "Lent"
        Lamp1 (14,146 70x70), variable: NTCProcess.bVagoHajlitoFent, style: Lamp-Lamp1-Yellow
        Label (24,120 50x30), "Fent"
        Label (131,31 69x30), "Kiszedö"
        Lamp1 (130,237 70x70), variable: NTCProcess.bKiszedoBent, style: Lamp-Lamp1-Yellow
        Label (146,211 38x30), "Bent"
        Lamp1 (130,146 70x70), variable: NTCProcess.bKiszedoKint, style: Lamp-Lamp1-Yellow
        Label (147,120 36x30), "Kint"
        PushSwitch (130,58 70x70), variable: NTCProcess.bKiszedo, behaviour: TOGGLE, style: Switch-PushSwitch-Red
        PushSwitch (249,58 70x70), variable: NTCProcess.bMegfogo, behaviour: TOGGLE, style: Switch-PushSwitch-Red
        Lamp1 (249,237 70x70), variable: NTCProcess.bMegfogoZarva, style: Lamp-Lamp1-Yellow
        Label (265,211 39x30), "Zárva"
        Lamp1 (249,146 70x70), variable: NTCProcess.bMegfogoNyitva, style: Lamp-Lamp1-Yellow
        Label (261,120 47x30), "Nyitva"
        Label (251,31 69x30), "Megfogó"
        Line (106,319) (106,38)
        Line (225,319) (225,38)
    RoundedRectangle (18,19 150x30)
    Label (18,20 150x30), "NTC-VÁGÓ"
    Group (194,8 131x70)
        PushSwitch (61,0 70x70), variable: MAIN.bLevego, behaviour: TOGGLE, style: Switch-PushSwitch-Red
        Label (0,20 55x30), "LEVEGÖ"
    Button (7,405 160x60), "NTC vágás"
        OnMouseClick: execute { NTCProcess.s_InCommand:='VAGAS'; }
    Button (183,405 160x60), "NTC elengedés"
        OnMouseClick: execute { NTCProcess.s_InCommand:='NTC_ELENGED'; }
    Rectangle (377,406 555x55)
    Checkbox (692,413 227x44), "Zöld gomb: NTC vágás Piros gomb: NTC elengedés", variable: NTC.bVagasGombbal, input disabled if: NTC.bVagoFelLeGombbal AND FALSE
    GroupBox (352,74 214x232), "NTC pozícionálás"
        Label (19,125 69x20), "Bal fék"
        Lamp1 (19,56 70x70), variable: NTC.bNTCLaberzekeloBal, style: Lamp-Lamp1-Yellow
        Label (4,35 99x20), "Bal lábérzékelö"
        PushSwitch (126,145 70x70), variable: NTC.bNTCFekJobb, behaviour: TOGGLE, style: Switch-PushSwitch-Red
    PushSwitch (369,219 70x70), variable: NTC.bNTCFekBal, behaviour: TOGGLE, style: Switch-PushSwitch-Red
    Label (480,199 69x20), "Jobb fék"
    Lamp1 (480,130 70x70), variable: NTC.bNTCLaberzekeloJobb, style: Lamp-Lamp1-Yellow
    Label (465,109 99x20), "Jobb lábérzékelö"
    Lamp1 (371,332 66x66), variable: NTC.bZoldGomb, style: Lamp-Lamp1-Green
    Lamp1 (481,332 66x66), variable: NTC.bPirosGomb, style: Lamp-Lamp1-Red
    Label (480,310 69x20), "Piros gomb"
    Label (370,310 69x20), "Zöld gomb"
    Checkbox (384,413 297x44), "Fizikális gombok használata NTC vágáshoz. Zöld gomb: NTC vágófej le-fel Piros gomb: NTC vágófej le-fel", variable: NTC.bVagoFelLeGombbal, input disabled if: TRUE
    Line (685,458) (685,408)
END_VISUALIZATION

// ---- VISUs/Hegesztok.TcVIS
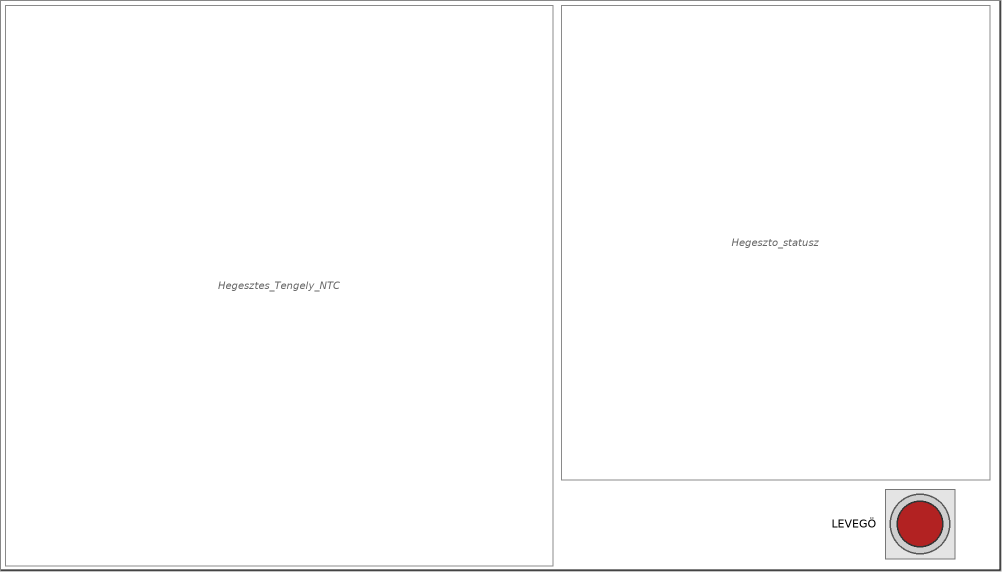
VISUALIZATION Hegesztok  // 1002x572
    Rectangle (0,0 1000x570)
    TabControl (5,5 548x561), frame switch variable: GVL.iTengelyLapozo
        shows Hegesztes_Tengely_NTC()
        shows Hegesztes_Tengely_Pt1000()
        shows Hegesztes_Karbantartas()
        [0]: TabTitle=NTC oldal
        [1]: TabTitle=Pt1000 oldal
        [2]: TabTitle=Elekróda karbantartás
    Group (824,489 131x70)
        PushSwitch (61,0 70x70), variable: MAIN.bLevego, behaviour: TOGGLE, style: Switch-PushSwitch-Red
        Label (0,20 55x30), "LEVEGÖ"
    TabControl (561,5 429x475)
        shows Hegeszto_statusz()
        shows Hegesztofej_IOk()
        shows Pt1000_oldali_kamera()
        [0]: TabTitle=Hegesztö státusz
        [1]: TabTitle=Hegesztöfej I/O-k
        [2]: TabTitle=Pt oldali kamera
END_VISUALIZATION

// ---- VISUs/Termeles0.TcVIS
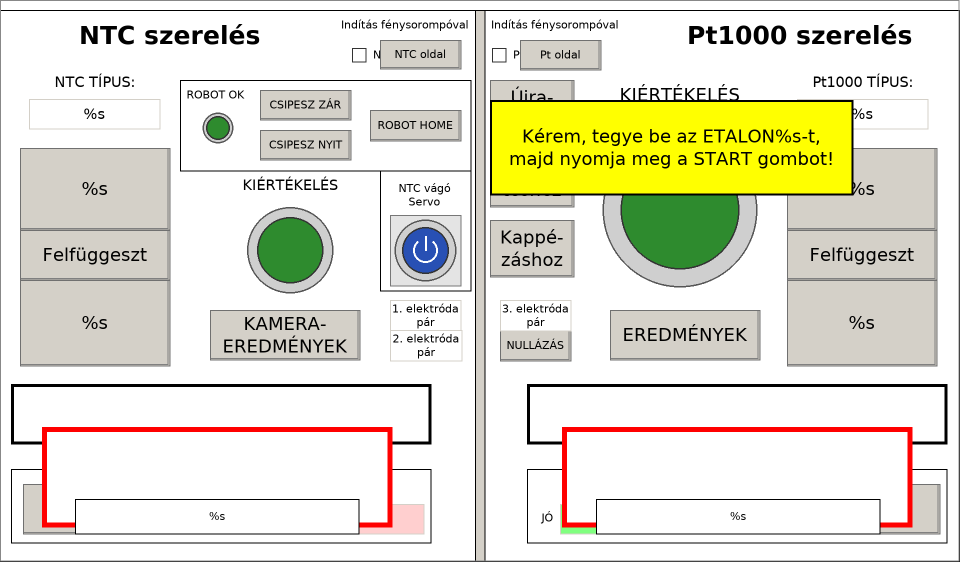
VISUALIZATION Termeles0  // 960x562
    Rectangle (0,10 960x552)
    Rectangle (380,170 91x121)
    Rectangle (180,80 291x91)
    RoundedRectangle (11,384 420x60), tooltip "Állapotváltozó: %s", text list: 'AUTOMATA_lepesek1', text index: AUTOMATA.iState
        p4168582468: AUTOMATA.iState
    Group (527,469 420x74)
        Rectangle (0,0 420x74)
        Textfield (33,35 81x30), "%s", text variable: GVL.nGoodProductCount
        Label (8,34 25x30), "JÓ"
        Textfield (170,35 81x30), "%s", text variable: GVL.nBadProductCount
        Label (128,34 42x30), "HIBÁS"
        Label (103,0 82x30), "DARABSZÁM"
        Button (263,15 150x50), "NULLÁZ"
            OnMouseUp: execute { GVL.nGoodProductCount:=0; GVL.nBadProductCount:=0; }
    RoundedRectangle (527,384 420x60), tooltip "Állapotváltozó: %s", text list: 'AUTOMATA_lepesek2', text index: AUTOMATA.iState2
        p4168582468: AUTOMATA.iState2
    Label (690,20 220x30), "Pt1000 szerelés"
    Group (590,80 180x220)
        Lamp1 (0,40 180x180), variable: GVL.bProductNOK, style: Lamp-Lamp1-Red
        Lamp1 (0,40 180x180), variable: GVL.bProductOK, invisible if: GVL.bProductNOK, style: Lamp-Lamp1-Green
        Label (0,0 180x30), "KIÉRTÉKELÉS"
    Button (787,148 150x82), "%s", text variable: AUTOMATA.sStart2GombFelirat, colour toggle: GVL.nElectrode3Usage>GVL.nElectrode3UsageWarn, input disabled if: NOT (ABS(PISTITENGELY.lrPistiActPos-GVL.lrPtSzervizbox)<0.1) AND NOT AUTOMATA.bContinue2En
        p573394764: GVL.nElectrode3AlarmColor
        OnMouseUp: execute {
            IF AUTOMATA.iState2=0 THEN
            	AUTOMATA.iState2:=1;
            ELSE
            	AUTOMATA.bContinue2:=TRUE;
            END_IF
        }
    Button (787,280 150x86), "%s", text variable: AUTOMATA.sStop2GombFelirat, input disabled if: (AUTOMATA.iState2=0) AND ABS(PISTITENGELY.lrPistiActPos-GVL.lrPtSzervizbox)<0.1
        OnMouseUp: execute {
            IF NOT(AUTOMATA.iState2=99) THEN
            //	AUTOMATA.bContinue2:=FALSE;
            //	AUTOMATA.bWelderReservedBy2:=FALSE;
            //	AUTOMATA.bRobotReservedBy2:=FALSE;
            //	GVL.bAdapterLefogo:=FALSE;
            //	AUTOMATA.sStop2GombFelirat:='Szervízboxhoz';
            //	AUTOMATA.bStart2GombTiltva:=TRUE;
            //	AUTOMATA.sStart2GombFelirat:='START';
            //	PISTITENGELY.sPistiAxisCommand:='STOP';
            //	AUTOMATA.iState2:=0;
            	AUTOMATA.iState2:=200;
            ELSE
            	AUTOMATA.iState2:=100;
            END_IF
        }
    Button (610,310 150x50), "EREDMÉNYEK"
        OnMouseUp: execute { GVL.bMeresiEredmenyekRejtve:=FALSE; }
    Group (11,469 420x74)
        Rectangle (0,0 420x74)
        Textfield (195,35 81x30), "%s", text variable: GVL.nGoodProductCount1
        Label (170,34 25x30), "JÓ"
        Textfield (332,35 81x30), "%s", text variable: GVL.nBadProductCount1
        Label (290,34 42x30), "HIBÁS"
        Label (265,0 82x30), "DARABSZÁM"
        Button (12,15 150x50), "NULLÁZ"
            OnMouseUp: execute { GVL.nGoodProductCount1:=0; GVL.nBadProductCount1:=0; }
    Button (20,148 150x82), "%s", text variable: AUTOMATA.sStart1GombFelirat, colour toggle: (GVL.nElectrode1Usage>GVL.nElectrode1UsageWarn) OR (GVL.nElectrode2Usage>GVL.nElectrode2UsageWarn), input disabled if: AUTOMATA.bStart1GombTiltva
        p573394764: MIN(GVL.nElectrode1AlarmColor,GVL.nElectrode2AlarmColor)
        OnMouseUp: execute {
            IF AUTOMATA.iState=0 THEN
            	AUTOMATA.iState:=1;
            ELSE
            	AUTOMATA.bContinue:=TRUE;
            END_IF
        }
    Button (20,280 150x86), "%s", text variable: AUTOMATA.sStop1GombFelirat, input disabled if: (AUTOMATA.iState=0) AND ABS(JOZSITENGELY.lrJozsiActPos-GVL.lrNTCSzervizbox)<0.1
        OnMouseUp: execute {
            AUTOMATA.bStopMegnyomva:=TRUE;
            //IF NOT(AUTOMATA.iState=0) THEN
            //	AUTOMATA.bContinue:=FALSE;
            //	AUTOMATA.bWelderReservedBy1:=FALSE;
            //	AUTOMATA.bRobotReservedBy1:=FALSE;
            //	JOZSITENGELY.sJozsiAxisCommand:='STOP';
            //	AUTOMATA.iState:=0;
            //	AUTOMATA.iState:=130;
            //ELSE
            //	AUTOMATA.iState:=100;
            //END_IF
        }
    Label (70,20 200x30), "NTC szerelés"
    Lamp1 (240,200 100x100), variable: GVL.bProduct1NOK, style: Lamp-Lamp1-Red
    Lamp1 (240,200 100x100), variable: GVL.bProduct1OK, invisible if: GVL.bProduct1NOK, style: Lamp-Lamp1-Green
    Label (220,170 141x30), "KIÉRTÉKELÉS"
    Rectangle (475,10 10x552)
    Label (40,67 110x30), "NTC TÍPUS:"
    Textfield (29,99 131x30), "%s", text variable: GVL.sNTCTypeElozo, colour toggle: GVL.sNTCType='HIBÁS KÓD'
        OnMouseClick: write GVL.sNTCType via Edit
    Label (808,67 110x30), "Pt1000 TÍPUS:"
    Textfield (797,99 131x30), "%s", text variable: GVL.sPtTypeElozo, colour toggle: GVL.sPtType='HIBÁS KÓD'
        OnMouseClick: write GVL.sPtType via Edit
    Button (490,80 84x57), "Újra- mérés", text variable: AUTOMATA.sStart2GombFelirat, colour toggle: AUTOMATA.bUjrameres, pressed state: AUTOMATA.bUjrameres, invisible if: TRUE
        OnMouseClick: execute {
            AUTOMATA.bUjrameres:=NOT AUTOMATA.bUjrameres;
            IF AUTOMATA.bUjrameres THEN
            	AUTOMATA.bHegesztes6Be:=GVL.bHegesztes6Be;
            	AUTOMATA.bHegesztes7Be := GVL.bHegesztes7Be;
            	AUTOMATA.bPtKameraBe := GVL.bPtKameraBe;
            	AUTOMATA.bRobotKappeBe := GVL.bRobotKappeBe;
            	AUTOMATA.bKappeBe := GVL.bKappeBe;
            	AUTOMATA.bMeresBe := GVL.bMeresBe;
            	AUTOMATA.bJelolesBe := GVL.bJelolesBe;
            	GVL.bHegesztes6Be := FALSE;
            	GVL.bHegesztes7Be := FALSE;
            	GVL.bPtKameraBe := FALSE;
            	GVL.bRobotKappeBe := FALSE;
            	GVL.bKappeBe := TRUE;
            	GVL.bMeresBe := TRUE;
            	GVL.bJelolesBe := TRUE;
            ELSE
            	GVL.bHegesztes6Be:=AUTOMATA.bHegesztes6Be;
            	GVL.bHegesztes7Be := AUTOMATA.bHegesztes7Be;
            	GVL.bPtKameraBe := AUTOMATA.bPtKameraBe;
            	GVL.bRobotKappeBe := AUTOMATA.bRobotKappeBe;
            	GVL.bKappeBe := AUTOMATA.bKappeBe;
            	GVL.bMeresBe := AUTOMATA.bMeresBe;
            	GVL.bJelolesBe := AUTOMATA.bJelolesBe;
            END_IF
        }
    Button (787,230 150x50), "Felfüggeszt", pressed state: AUTOMATA.bFelfuggeszt2
        OnMouseUp: execute {
            IF AUTOMATA.bFelfuggeszt2=FALSE THEN
            	AUTOMATA.bFelfuggeszt2:=TRUE;
            	AUTOMATA.iState2Elozo:=AUTOMATA.iState2;
            	AUTOMATA.iState2:=300;
            ELSE
            	AUTOMATA.bFelfuggeszt2:=FALSE;
            END_IF
        }
    Button (20,230 150x50), "Felfüggeszt", pressed state: AUTOMATA.bFelfuggeszt
        OnMouseUp: execute {
            IF AUTOMATA.bFelfuggeszt=FALSE THEN
            	AUTOMATA.bFelfuggeszt:=TRUE;
            	AUTOMATA.iStateElozo:=AUTOMATA.iState;
            	AUTOMATA.iState:=300;
            ELSE
            	AUTOMATA.bFelfuggeszt:=FALSE;
            END_IF
        }
    Group (42,427 350x107)
        RoundedRectangle (0,0 350x100), invisible if: GVL.bHibauzenetNTCRejtve, text list: 'ErrorList', text index: GVL.nHibaKodNTC
        Rectangle (33,72 284x35), "%s", text variable: AUTOMATA.sRobotHiba, invisible if: GVL.bHibauzenetNTCRejtve OR NOT (GVL.nHibaKodNTC=307)
    Group (562,427 350x107)
        RoundedRectangle (0,0 350x100), invisible if: GVL.bHibauzenetPtRejtve, text list: 'ErrorList', text index: GVL.nHibaKodPt
        Rectangle (34,72 284x35), "%s", text variable: AUTOMATA.sRobotHiba, invisible if: GVL.bHibauzenetPtRejtve OR NOT (GVL.nHibaKodPt=307)
    Button (210,310 150x50), "KAMERA- EREDMÉNYEK"
        OnMouseUp: execute {
            GVL.bNTCBezarGombRejtve:=FALSE;
            GVL.bKameraEredmenyekRejtve:=FALSE;
            GVL.iBitmap_Version:=GVL.iBitmap_Version+1;
        }
    Button (490,150 84x57), "Hegesz- téshez", invisible if: (GVL.bPtKameraBe=TRUE) AND (AUTOMATA.bPtKameraGombokEnged=FALSE)
        tap AUTOMATA.bHegeszteshezGomb
    Button (490,220 84x57), "Kappé- záshoz", invisible if: (GVL.bPtKameraBe=TRUE) AND (AUTOMATA.bPtKameraGombokEnged=FALSE)
        tap AUTOMATA.bKappezashozGomb
    RoundedRectangle (490,100 363x95), "Kérem, tegye be az ETALON%s-t, majd nyomja meg a START gombot!", text variable: GVL.iCurrentProductType+4, invisible if: NOT (GVL.iCurrentProductType<0) OR NOT GVL.bMeresBe
    Label (180,80 71x30), "ROBOT OK", invisible if: ROBOTREMOTE.bRobotCommOpen=FALSE
    Lamp1 (200,110 36x36), variable: RobotProcess.baStatus[9], invisible if: ROBOTREMOTE.bRobotCommOpen=FALSE, style: Lamp-Lamp1-Green
    Checkbox (350,40 95x30), "NTC oldal", variable: GVL.bNTCInditasFenysorompoval, input disabled if: TRUE
    Checkbox (490,40 95x30), "Pt oldal", variable: GVL.bPtInditasFenysorompoval, input disabled if: TRUE
    Label (330,10 150x30), "Indítás fénysorompóval"
    Label (480,10 150x30), "Indítás fénysorompóval"
    Button (520,40 81x30), "Pt oldal", pressed state: GVL.bPtInditasFenysorompoval
        toggle GVL.bPtInditasFenysorompoval
        OnMouseUp: execute { AUTOMATA.iState2:=103; }
    Button (380,40 81x29), "NTC oldal", pressed state: GVL.bNTCInditasFenysorompoval
        toggle GVL.bNTCInditasFenysorompoval
        OnMouseUp: execute { AUTOMATA.iState:=102; }
    Textfield (390,300 71x31), "1. elektróda pár", text variable: GVL.nElectrode1Usage, colour toggle: GVL.nElectrode1Usage>GVL.nElectrode1UsageWarn
        p2167032090: GVL.nElectrode1AlarmColor
    Textfield (390,330 72x31), "2. elektróda pár", text variable: GVL.nElectrode2Usage, colour toggle: GVL.nElectrode2Usage>GVL.nElectrode2UsageWarn
        p2167032090: GVL.nElectrode2AlarmColor
    Button (500,330 71x31), "NULLÁZÁS"
        OnMouseUp: execute { GVL.nElectrode3Usage:=0; }
    Textfield (500,300 71x31), "3. elektróda pár", text variable: GVL.nElectrode3Usage, colour toggle: GVL.nElectrode3Usage>GVL.nElectrode3UsageWarn
        p2167032090: GVL.nElectrode3AlarmColor
    PowerSwitch (390,210 71x81), variable: NTC.bServoON, behaviour: TOGGLE, style: Switch-PowerSwitch-Blue
    Label (390,180 69x30), "NTC vágó Servo"
    Button (260,90 91x30), "CSIPESZ ZÁR", invisible if: RobotProcess.iState=0, input disabled if: RobotProcess.iState=0
        OnMouseClick: execute { RobotProcess.s_InRobotTCPCommand := 'CSIPESZ_ZAR'; }
    Button (260,130 91x30), "CSIPESZ NYIT", invisible if: RobotProcess.iState=0, input disabled if: RobotProcess.iState=0
        OnMouseClick: execute { RobotProcess.s_InRobotTCPCommand := 'CSIPESZ_NYIT'; }
    Button (370,110 91x31), "ROBOT HOME", invisible if: RobotProcess.iState=0, input disabled if: RobotProcess.iState=0
        OnMouseClick: execute { RobotProcess.s_InRobotTCPCommand := 'HOME'; }
END_VISUALIZATION

// ---- VISUs/Meresek.TcVIS
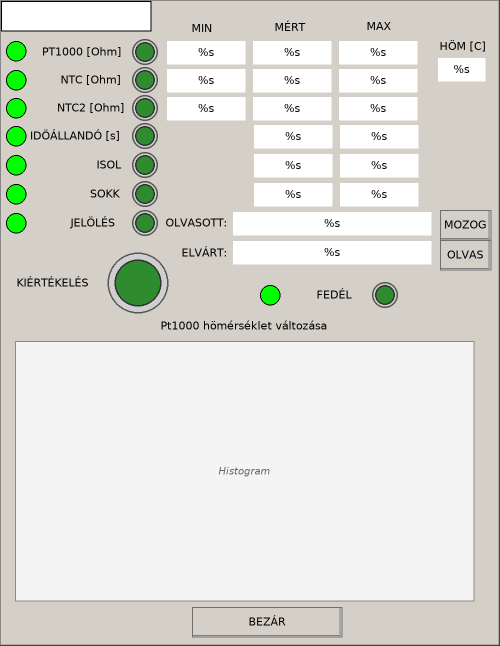
VISUALIZATION Meresek  // 500x646
    Rectangle (0,0 500x646)
    Lamp1 (130,150 30x30), variable: NOT GVL.bIsolOK, style: Lamp-Lamp1-Red
    Label (92,155 34x20), "ISOL"
    Label (182,16 40x25), "MIN"
    Histogram (15,341 459x260), scale format: %.1f, scale 0..300
        p1518820177: VEGMERO.arIdoallandoPTTEMP
        p102497268: VEGMERO.arIdoallandoPTTEMP
        p788070771: ARRAY [0..600] OF REAL
    Lamp1 (130,179 30x30), variable: NOT GVL.bShockOK, style: Lamp-Lamp1-Red
    Label (84,184 42x20), "SOKK"
    Label (60,213 66x20), "JELÖLÉS"
    Lamp1 (130,208 30x30), variable: NOT GVL.bMarkingOK, style: Lamp-Lamp1-Red
    Lamp1 (103,248 70x70), variable: GVL.bProductNOK, style: Lamp-Lamp1-Red
    Lamp1 (103,248 70x70), variable: GVL.bProductOK, invisible if: GVL.bProductNOK, style: Lamp-Lamp1-Green
    Label (7,268 91x30), "KIÉRTÉKELÉS"
    Label (38,42 88x20), "PT1000 [Ohm]"
    Lamp1 (130,37 30x30), variable: NOT GVL.bPTResOK, style: Lamp-Lamp1-Red
    Textfield (252,40 80x25), "%s", text variable: GVL.rPtRes
    Textfield (166,40 80x25), "%s", text variable: VEGMERO.PTRES_MIN
    Textfield (338,40 80x25), "%s", text variable: VEGMERO.PTRES_MAX
    Label (56,70 70x20), "NTC [Ohm]"
    Lamp1 (130,65 30x30), variable: NOT GVL.bNTCResOK, style: Lamp-Lamp1-Red
    Textfield (252,68 80x25), "%s", text variable: GVL.rNTCRes
    Textfield (166,68 80x25), "%s", text variable: VEGMERO.NTCRES_MIN
    Textfield (338,68 80x25), "%s", text variable: VEGMERO.NTCRES_MAX
    Lamp1 (130,121 30x30), variable: NOT GVL.bTimeConstOK, style: Lamp-Lamp1-Red
    Label (24,126 102x20), "IDÖÁLLANDÓ [s]"
    Textfield (253,124 80x25), "%s", text variable: GVL.rTimeConst
    Textfield (437,57 49x25), "%s", text variable: GVL.rTemp
    Label (359,14 40x25), "MAX"
    Label (270,15 40x25), "MÉRT"
    Label (438,34 50x25), "HÖM [C]"
    Textfield (339,124 80x25), "%s", text variable: REAL_TO_TIME(GVL.rIdoallandoMax*1000)
    Label (144,311 200x30), "Pt1000 hömérséklet változása"
    Textfield (253,153 80x25), "%s", text variable: VEGMERO.rISOL
    Textfield (339,153 80x25), "%s", text variable: GVL.rISOL_MAX
    Textfield (232,211 200x25), "%s", text variable: ZEBRASCANNER.sReceivedString255
    Button (192,607 150x30), "BEZÁR", invisible if: GVL.bMeresiEredmenyekRejtve
        OnMouseUp: execute { GVL.bMeresiEredmenyekRejtve:=TRUE; }
    Textfield (232,240 200x25), "%s", text variable: AUTOMATA.sExpectedCode
    Label (164,213 66x20), "OLVASOTT:"
    Label (164,243 66x20), "ELVÁRT:"
    Textfield (253,182 80x25), "%s", text variable: GVL.rPtResShock
    Textfield (339,182 80x25), "%s", text variable: GVL.PTRES_SOKK_MAX
    Lamp1 (130,37 30x30), variable: GVL.bPTResOK, invisible if: NOT GVL.bPTResOK AND VEGMERO.bPTRES_MERVE, style: Lamp-Lamp1-Green
    Lamp1 (130,150 30x30), variable: GVL.bIsolOK, invisible if: NOT GVL.bIsolOK AND VEGMERO.bISOL_MERVE, style: Lamp-Lamp1-Green
    Lamp1 (130,179 30x30), variable: GVL.bShockOK, invisible if: NOT GVL.bShockOK AND VEGMERO.bSOKK_MERVE, style: Lamp-Lamp1-Green
    Lamp1 (130,208 30x30), variable: GVL.bMarkingOK, invisible if: NOT GVL.bMarkingOK AND GVL.bMarking_ellenorizve, style: Lamp-Lamp1-Green
    Lamp1 (130,65 30x30), variable: GVL.bNTCResOK, invisible if: NOT GVL.bNTCResOK AND VEGMERO.bNTCRES_MERVE, style: Lamp-Lamp1-Green
    Lamp1 (130,121 30x30), variable: GVL.bTimeConstOK, invisible if: NOT GVL.bTimeConstOK AND VEGMERO.bIDOALLANDO_MERVE, style: Lamp-Lamp1-Green
    Ellipse (6,41 20x20), colour toggle: AUTOMATA.iProductTypeUnderTest<-1, invisible if: NOT GVL.bMeresBe
    Ellipse (6,70 20x20), colour toggle: AUTOMATA.iProductTypeUnderTest<-1, invisible if: NOT GVL.bMeresBe
    Ellipse (6,126 20x20), invisible if: (AUTOMATA.iProductTypeUnderTest<-1) OR NOT GVL.bMeresBe
    Ellipse (6,155 20x20), colour toggle: AUTOMATA.iProductTypeUnderTest=-2, invisible if: NOT GVL.bMeresBe
    Ellipse (6,213 20x20), invisible if: NOT GVL.bMeresBe
    Ellipse (6,184 20x20), invisible if: (AUTOMATA.iProductTypeUnderTest<0) OR NOT GVL.bMeresBe
    Label (290,285 88x20), "FEDÉL"
    Lamp1 (370,280 30x30), variable: GVL.bFedelOK OR GVL.bHimbaOK, style: Lamp-Lamp1-Green
    Ellipse (260,285 20x20), colour toggle: AUTOMATA.iProductTypeUnderTest<-2, invisible if: NOT GVL.bMeresBe
    Rectangle (1,1 150x30), text list: 'DUT_types', text index: GVL.iCurrentProductType+3
    Ellipse (6,98 20x20), colour toggle: AUTOMATA.iProductTypeUnderTest<-1, invisible if: NOT GVL.bMeresBe OR (GVL.iSelectedProductType<8)
    Label (56,98 70x20), "NTC2 [Ohm]"
    Textfield (252,96 80x25), "%s", text variable: GVL.rNTCRes2
    Textfield (166,96 80x25), "%s", text variable: VEGMERO.NTCRES2_MIN
    Textfield (338,96 80x25), "%s", text variable: VEGMERO.NTCRES2_MAX
    Lamp1 (130,93 30x30), variable: NOT GVL.bNTCRes2OK, style: Lamp-Lamp1-Red
    Lamp1 (130,93 30x30), variable: GVL.bNTCRes2OK, invisible if: NOT GVL.bNTCRes2OK AND VEGMERO.bNTCRES2_MERVE, style: Lamp-Lamp1-Green
    Button (440,210 51x30), "MOZOG"
        OnMouseUp: execute { PISTITENGELY.lrPistiPosition:=GVL.lrKodolvasasPosition; PISTITENGELY.sPistiAxisCommand:='MOVE'; }
    Button (440,240 51x30), "OLVAS"
        OnMouseUp: execute { ZEBRASCANNER.bStartSend:=true; }
END_VISUALIZATION

// ---- VISUs/Beallitasok.TcVIS
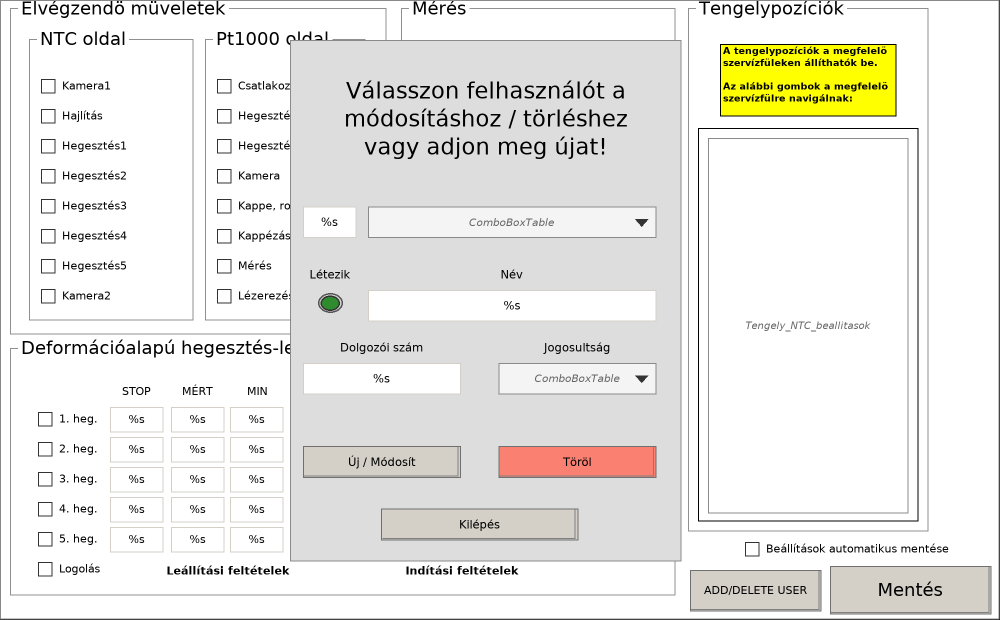
VISUALIZATION Beallitasok  // 1000x620
    Rectangle (0,0 1000x620)
    GroupBox (10,0 376x334), "Elvégzendö müveletek", invisible if: GVL.UserActual.UserLevel<1, input disabled if: GVL.UserActual.UserLevel<2
        GroupBox (19,31 164x289), "NTC oldal"
            Checkbox (10,70 140x30), "Hajlítás", variable: GVL.bHajlitasBe, input disabled if: AUTOMATA.bFolyamatBeallitas1Tiltva
            Checkbox (10,100 140x30), "Hegesztés1", variable: GVL.bHegesztes1Be, input disabled if: AUTOMATA.bFolyamatBeallitas1Tiltva
            Checkbox (10,130 140x30), "Hegesztés2", variable: GVL.bHegesztes2Be, input disabled if: AUTOMATA.bFolyamatBeallitas1Tiltva
            Checkbox (10,160 140x30), "Hegesztés3", variable: GVL.bHegesztes3Be, input disabled if: AUTOMATA.bFolyamatBeallitas1Tiltva
            Checkbox (10,190 140x30), "Hegesztés4", variable: GVL.bHegesztes4Be, input disabled if: AUTOMATA.bFolyamatBeallitas1Tiltva
            Checkbox (10,220 140x30), "Hegesztés5", variable: GVL.bHegesztes5Be, input disabled if: AUTOMATA.bFolyamatBeallitas1Tiltva
            Checkbox (10,40 140x30), "Kamera1", variable: GVL.bKameraBe, input disabled if: AUTOMATA.bFolyamatBeallitas1Tiltva
            Checkbox (10,250 140x30), "Kamera2", variable: GVL.bKameraVegBe, input disabled if: AUTOMATA.bFolyamatBeallitas1Tiltva
        GroupBox (195,31 160x289), "Pt1000 oldal"
            Checkbox (10,250 140x30), "Lézerezés", variable: GVL.bJelolesBe, input disabled if: AUTOMATA.bFolyamatBeallitas2Tiltva
            Checkbox (10,70 140x30), "Hegesztés1", variable: GVL.bHegesztes6Be, input disabled if: AUTOMATA.bFolyamatBeallitas2Tiltva
            Checkbox (10,100 140x30), "Hegesztés2", variable: GVL.bHegesztes7Be, input disabled if: AUTOMATA.bFolyamatBeallitas2Tiltva
            Checkbox (10,160 140x30), "Kappe, robot", variable: GVL.bRobotKappeBe, input disabled if: AUTOMATA.bFolyamatBeallitas2Tiltva
            Checkbox (10,190 140x30), "Kappézás", variable: GVL.bKappeBe, input disabled if: AUTOMATA.bFolyamatBeallitas2Tiltva
            Checkbox (10,220 140x30), "Mérés", variable: GVL.bMeresBe, input disabled if: AUTOMATA.bFolyamatBeallitas2Tiltva
            Checkbox (10,130 140x30), "Kamera", variable: GVL.bPtKameraBe, input disabled if: AUTOMATA.bFolyamatBeallitas2Tiltva AND TRUE
            Checkbox (10,40 140x30), "Csatlakozó (745)", variable: GVL.bHimbaBe, input disabled if: AUTOMATA.bFolyamatBeallitas2Tiltva AND (GVL.iSelectedProductType<=8)
    GroupBox (401,0 274x334), "Mérés", invisible if: GVL.UserActual.UserLevel<1, input disabled if: GVL.UserActual.UserLevel<2
        Checkbox (30,43 116x30), "Etalon mérés", variable: GVL.bEtalonOn
        Textfield (136,83 120x30), "%s", text variable: GVL.rNTCDev
            OnMouseClick: write the text variable via VisuDialogs.Numpad, min 0, max 30
        Label (42,83 89x30), "NTC1 türés [%]:"
        Textfield (136,188 120x30), "%s", text variable: GVL.rISOL_MAX
            OnMouseUp: write the text variable via VisuDialogs.Numpad, min 0, max 2
        Label (34,187 93x30), "Max. szigetelési érték [V]:"
        Textfield (136,223 120x30), "%f", text variable: GVL.rTempMax
            OnMouseClick: write the text variable via VisuDialogs.Numpad, min 0, max 400
        Label (54,257 73x30), "Idöállandó felsö határa [s]:"
        Textfield (136,258 120x30), "%s", text variable: GVL.rIdoallandoMax
            OnMouseClick: write the text variable via VisuDialogs.Numpad, min 0, max 8
        Textfield (136,153 120x30), "%s", text variable: GVL.rPtDev
            OnMouseClick: write the text variable via VisuDialogs.Numpad, min 0, max 15
        Label (27,152 104x30), "Pt1000 türés [%]:"
        Textfield (136,293 120x30), "%s", text variable: GVL.PTRES_SOKK_MAX
            OnMouseClick: write the text variable via VisuDialogs.Numpad, min 0, max 3000
        Label (22,222 106x34), "Fütötömb beállított hömérséklete [C]:"
        Label (11,292 114x30), "Sokkolás, max Pt ellenállás [Ohm]:"
        Label (42,117 89x30), "NTC2 türés [%]:"
        Textfield (136,118 120x30), "%s", text variable: GVL.rNTC2Dev
            OnMouseClick: write the text variable via VisuDialogs.Numpad, min 0, max 30
    GroupBox (688,0 240x531), "Tengelypozíciók", invisible if: GVL.UserActual.UserLevel<1, input disabled if: GVL.UserActual.UserLevel<2
        Rectangle (32,44 176x72), "A tengelypozíciók a megfelelö szervízfüleken állíthatók be. Az alábbi gombok a megfelelö szervízfülre navigálnak:"
        Rectangle (10,128 220x393)
        TabControl (20,138 200x375)
            shows Tengely_NTC_beallitasok()
            shows Tengely_Pt1000_beallitasok()
            [0]: TabTitle=NTC oldal
            [1]: TabTitle=Pt1000 oldal
    GroupBox (10,340 665x255), "Deformációalapú hegesztés-leállítás", invisible if: GVL.UserActual.UserLevel<1, input disabled if: GVL.UserActual.UserLevel<2
        Checkbox (26,154 75x30), "4. heg.", variable: GVL.bAutomaticWeldingStop4
        Checkbox (26,184 75x30), "5. heg.", variable: GVL.bAutomaticWeldingStop5
        Checkbox (26,124 75x30), "3. heg.", variable: GVL.bAutomaticWeldingStop3
        Checkbox (26,94 75x30), "2. heg.", variable: GVL.bAutomaticWeldingStop2
        Checkbox (26,64 75x30), "1. heg.", variable: GVL.bAutomaticWeldingStop1
        Textfield (100,187 53x25), "%s", text variable: GVL.nWeldingStopDistance5
            OnMouseClick: write the text variable via VisuDialogs.Numpad, min 0, max 1000
        Textfield (100,157 53x25), "%s", text variable: GVL.nWeldingStopDistance4
            OnMouseClick: write the text variable via VisuDialogs.Numpad, min 0, max 1000
        Textfield (100,127 53x25), "%s", text variable: GVL.nWeldingStopDistance3
            OnMouseClick: write the text variable via VisuDialogs.Numpad, min 0, max 1000
        Textfield (100,97 53x25), "%s", text variable: GVL.nWeldingStopDistance2
            OnMouseClick: write the text variable via VisuDialogs.Numpad, min 0, max 1000
        Textfield (100,67 53x25), "%s", text variable: GVL.nWeldingStopDistance1
            OnMouseClick: write the text variable via VisuDialogs.Numpad, min 0, max 1000
        Textfield (161,67 53x25), "%s", text variable: GVL.nWeldingDeformation1
        Textfield (161,97 53x25), "%s", text variable: GVL.nWeldingDeformation2
        Textfield (161,127 53x25), "%s", text variable: GVL.nWeldingDeformation3
        Textfield (161,157 53x25), "%s", text variable: GVL.nWeldingDeformation4
        Textfield (161,187 53x25), "%s", text variable: GVL.nWeldingDeformation5
        Label (104,39 45x25), "STOP"
        Label (165,39 45x25), "MÉRT"
        Checkbox (26,214 87x30), "Logolás", variable: GVL.bWeldingLog
        Label (342,67 25x25), "um"
        Label (342,97 25x25), "um"
        Label (342,127 25x25), "um"
        Label (342,157 25x25), "um"
        Label (342,187 25x25), "um"
        Textfield (220,67 53x25), "%s", text variable: GVL.nWeldingDistanceMin1
            OnMouseClick: write the text variable via VisuDialogs.Numpad, min 0, max 2000
        Label (225,39 45x25), "MIN"
        Label (143,216 150x30), "Leállítási feltételek"
        Label (377,216 150x30), "Indítási feltételek"
        Textfield (370,97 53x25), "%s", text variable: GVL.ulWeldingStartDistance2
        Textfield (370,127 53x25), "%s", text variable: GVL.ulWeldingStartDistance3
        Textfield (370,187 53x25), "%s", text variable: GVL.ulWeldingStartDistance5
        Textfield (280,67 53x25), "%s", text variable: GVL.nWeldingDistanceMax1
            OnMouseClick: write the text variable via VisuDialogs.Numpad, min 0, max 2000
        Textfield (280,97 53x25), "%s", text variable: GVL.nWeldingDistanceMax2
            OnMouseClick: write the text variable via VisuDialogs.Numpad, min 0, max 2000
        Textfield (220,97 53x25), "%s", text variable: GVL.nWeldingDistanceMin2
            OnMouseClick: write the text variable via VisuDialogs.Numpad, min 0, max 2000
        Textfield (220,127 53x25), "%s", text variable: GVL.nWeldingDistanceMin3
            OnMouseClick: write the text variable via VisuDialogs.Numpad, min 0, max 2000
        Textfield (220,157 53x25), "%s", text variable: GVL.nWeldingDistanceMin4
            OnMouseClick: write the text variable via VisuDialogs.Numpad, min 0, max 2000
        Textfield (220,187 53x25), "%s", text variable: GVL.nWeldingDistanceMin5
            OnMouseClick: write the text variable via VisuDialogs.Numpad, min 0, max 2000
        Textfield (280,187 53x25), "%s", text variable: GVL.nWeldingDistanceMax5
            OnMouseClick: write the text variable via VisuDialogs.Numpad, min 0, max 2000
        Textfield (280,157 53x25), "%s", text variable: GVL.nWeldingDistanceMax4
            OnMouseClick: write the text variable via VisuDialogs.Numpad, min 0, max 2000
        Textfield (280,127 53x25), "%s", text variable: GVL.nWeldingDistanceMax3
            OnMouseClick: write the text variable via VisuDialogs.Numpad, min 0, max 2000
        Textfield (370,67 53x25), "%s", text variable: GVL.ulWeldingStartDistance1
        Textfield (370,157 53x25), "%s", text variable: GVL.ulWeldingStartDistance4
        Textfield (430,67 53x25), "%s", text variable: GVL.nWeldingDistanceStartMin1
            OnMouseClick: write the text variable via VisuDialogs.Numpad, min 0, max 200000
        Textfield (430,187 53x25), "%s", text variable: GVL.nWeldingDistanceStartMin5
            OnMouseClick: write the text variable via VisuDialogs.Numpad, min 0, max 200000
        Textfield (430,157 53x25), "%s", text variable: GVL.nWeldingDistanceStartMin4
            OnMouseClick: write the text variable via VisuDialogs.Numpad, min 0, max 200000
        Textfield (430,127 53x25), "%s", text variable: GVL.nWeldingDistanceStartMin3
            OnMouseClick: write the text variable via VisuDialogs.Numpad, min 0, max 200000
        Textfield (430,97 53x25), "%s", text variable: GVL.nWeldingDistanceStartMin2
            OnMouseClick: write the text variable via VisuDialogs.Numpad, min 0, max 200000
        Textfield (491,67 53x25), "%s", text variable: GVL.nWeldingDistanceStartMax1
            OnMouseClick: write the text variable via VisuDialogs.Numpad, min 0, max 210000
        Textfield (491,97 53x25), "%s", text variable: GVL.nWeldingDistanceStartMax2
            OnMouseClick: write the text variable via VisuDialogs.Numpad, min 0, max 210000
        Textfield (491,127 53x25), "%s", text variable: GVL.nWeldingDistanceStartMax3
            OnMouseClick: write the text variable via VisuDialogs.Numpad, min 0, max 210000
        Textfield (491,157 53x25), "%s", text variable: GVL.nWeldingDistanceStartMax4
            OnMouseClick: write the text variable via VisuDialogs.Numpad, min 0, max 210000
        Textfield (491,187 53x25), "%s", text variable: GVL.nWeldingDistanceStartMax5
            OnMouseClick: write the text variable via VisuDialogs.Numpad, min 0, max 210000
        Label (550,100 25x25), "um"
        Label (550,70 25x25), "um"
        Label (550,130 25x25), "um"
        Label (550,160 25x25), "um"
        Label (550,190 25x25), "um"
        Label (283,40 45x25), "MAX"
        Label (377,40 45x25), "MÉRT"
        Label (433,40 45x25), "MIN"
        Label (493,40 45x25), "MAX"
    Checkbox (743,534 223x30), "Beállítások automatikus mentése", variable: GVL.bSettingsAutoSave, invisible if: GVL.UserActual.UserLevel<1, input disabled if: GVL.UserActual.UserLevel<2
    Button (830,566 161x48), "Mentés", invisible if: GVL.UserActual.UserLevel<1, input disabled if: GVL.UserActual.UserLevel<2
        OnMouseClick: execute { MAIN.iStateS:=3; }
    Button (690,570 131x41), "ADD/DELETE USER", invisible if: GVL.UserActual.UserLevel<3, input disabled if: GVL.AddDelButtonDis
        toggle GVL.AddDeleteEnabled
    Frame (290,40 391x521), invisible if: NOT GVL.AddDeleteEnabled
        shows AddDelete()
END_VISUALIZATION

// ---- VISUs/Vegmero_idoallando.TcVIS
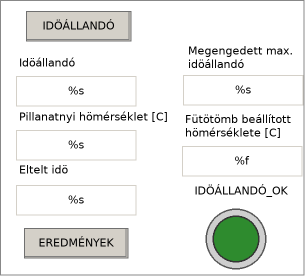
VISUALIZATION Vegmero_idoallando  // 305x276
    Button (26,11 105x30), "IDÖÁLLANDÓ", input disabled if: VEGMERO.s_InCommand<>''
        OnMouseUp: execute { VEGMERO.s_InCommand:='IDOALLANDO'; }
    Textfield (16,76 120x30), "%s", text variable: VEGMERO.tIdoallando
    Textfield (16,130 120x30), "%s", text variable: VEGMERO.arIdoallandoPTTEMP[VEGMERO.nI]
    Textfield (16,185 120x30), "%s", text variable: VEGMERO.atIdoallando[VEGMERO.nI]
    Label (16,53 87x20), "Idöállandó"
    Label (16,107 164x20), "Pillanatnyi hömérséklet [C]"
    Label (16,160 89x20), "Eltelt idö"
    Lamp1 (201,204 70x70), variable: NOT VEGMERO.bIDOALLANDO_OK, style: Lamp-Lamp1-Red
    Label (186,181 110x20), "IDÖÁLLANDÓ_OK"
    Textfield (182,146 120x30), "%f", text variable: GVL.rTempMax
    Label (182,109 117x34), "Fütötömb beállított hömérséklete [C]"
    Textfield (183,75 120x30), "%s", text variable: REAL_TO_TIME(GVL.rIdoallandoMax*1000)
    Label (185,43 107x29), "Megengedett max. idöállandó"
    Lamp1 (201,204 70x70), variable: VEGMERO.bIDOALLANDO_OK, invisible if: NOT VEGMERO.bIDOALLANDO_OK AND VEGMERO.bIDOALLANDO_MERVE, style: Lamp-Lamp1-Green
    Button (24,228 104x30), "EREDMÉNYEK"
        OnMouseUp: execute { GVL.bMeresiEredmenyekRejtve:=FALSE; }
END_VISUALIZATION

// ---- VISUs/Vegmero_sokk.TcVIS
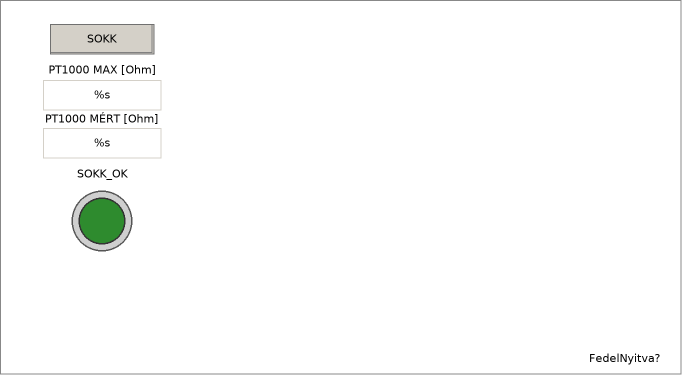
VISUALIZATION Vegmero_sokk  // 682x375
    Label (570,344 110x29), "FedelNyitva?"
    Textfield (43,128 118x30), "%s", text variable: VEGMERO.rPTRES
    Textfield (43,80 118x30), "%s", text variable: GVL.PTRES_SOKK_MAX
    Label (35,109 134x20), "PT1000 MÉRT [Ohm]"
    Label (39,60 127x20), "PT1000 MAX [Ohm]"
    Button (50,24 104x30), "SOKK", input disabled if: VEGMERO.s_InCommand<>''
        OnMouseUp: execute { VEGMERO.s_InCommand:='SOKK'; }
    Lamp1 (67,186 70x70), variable: NOT GVL.bShockOK, style: Lamp-Lamp1-Red
    Label (70,164 65x20), "SOKK_OK"
    Lamp1 (67,186 70x70), variable: GVL.bShockOK, invisible if: NOT GVL.bShockOK AND VEGMERO.bSOKK_MERVE, style: Lamp-Lamp1-Green
END_VISUALIZATION

// ---- VISUs/Vegmero_teljes.TcVIS
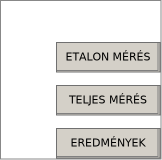
VISUALIZATION Vegmero_teljes  // 162x160
    Button (56,85 104x30), "TELJES MÉRÉS", input disabled if: VEGMERO.s_InCommand<>''
        OnMouseUp: execute { VEGMERO.s_InCommand:='TELJESMERES'; GVL.bMeresiEredmenyekRejtve:=FALSE; }
    Button (56,128 104x30), "EREDMÉNYEK"
        OnMouseUp: execute { GVL.bMeresiEredmenyekRejtve:=FALSE; }
    Button (56,42 104x30), "ETALON MÉRÉS", input disabled if: VEGMERO.s_InCommand<>''
        OnMouseUp: execute { VEGMERO.s_InCommand:='ETALONMERES'; GVL.bMeresiEredmenyekRejtve:=FALSE; }
END_VISUALIZATION

// ---- VISUs/Vegmero_szigeteles.TcVIS
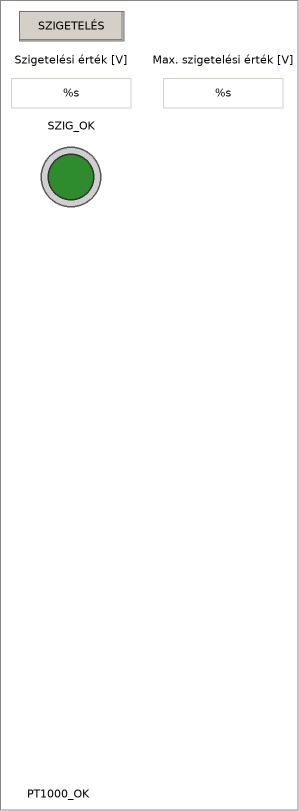
VISUALIZATION Vegmero_szigeteles  // 299x811
    Lamp1 (36,142 70x70), variable: NOT VEGMERO.bISOL_OK, style: Lamp-Lamp1-Red
    Label (36,116 70x20), "SZIG_OK"
    Button (19,11 105x30), "SZIGETELÉS", input disabled if: VEGMERO.s_InCommand<>''
        OnMouseUp: execute { VEGMERO.s_InCommand:='ATUTES'; }
    Textfield (11,78 120x30), "%s", text variable: VEGMERO.rISOL
    Label (11,50 120x20), "Szigetelési érték [V]"
    Label (3,779 110x30), "PT1000_OK"
    Textfield (163,78 120x30), "%s", text variable: GVL.rISOL_MAX
    Label (149,50 148x20), "Max. szigetelési érték [V]"
    Lamp1 (36,142 70x70), variable: VEGMERO.bISOL_OK, invisible if: NOT VEGMERO.bISOL_OK AND VEGMERO.bISOL_MERVE, style: Lamp-Lamp1-Green
END_VISUALIZATION

// ---- VISUs/Vegmero_auto.TcVIS
